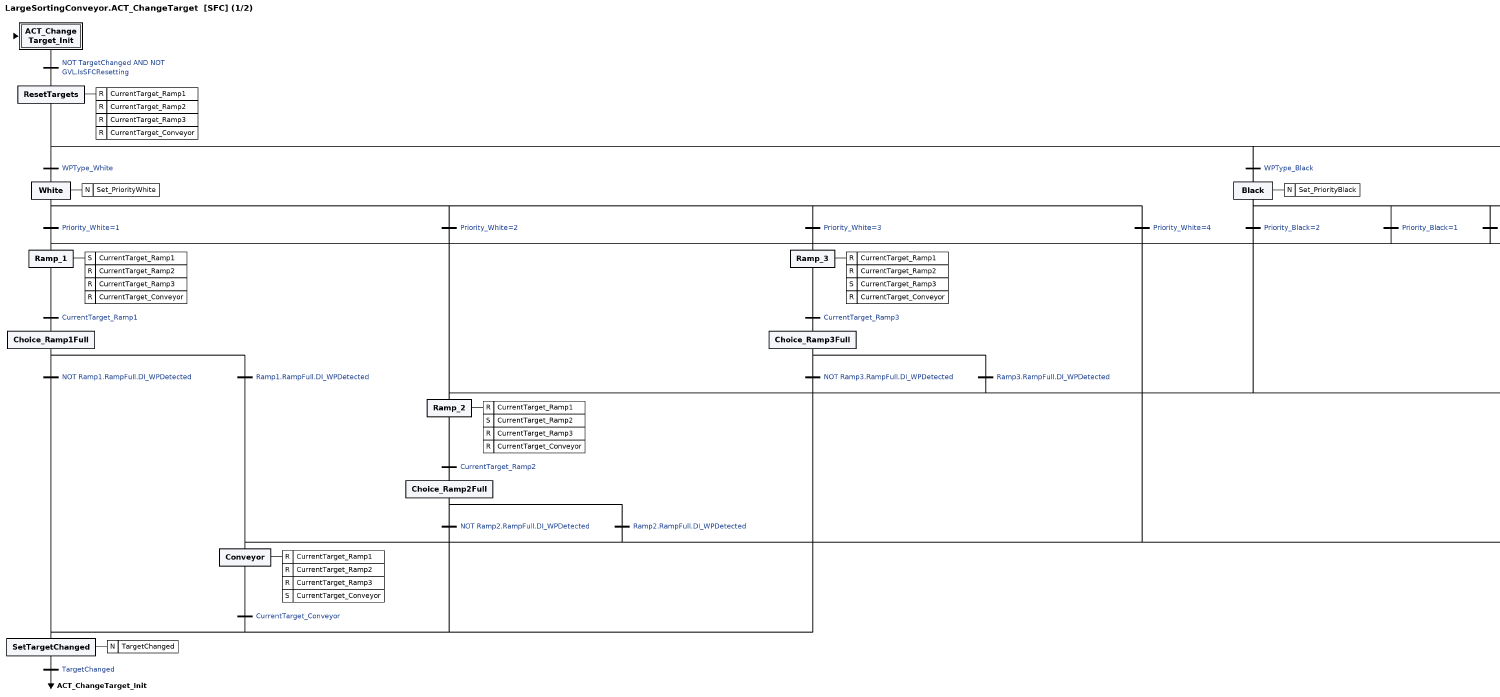
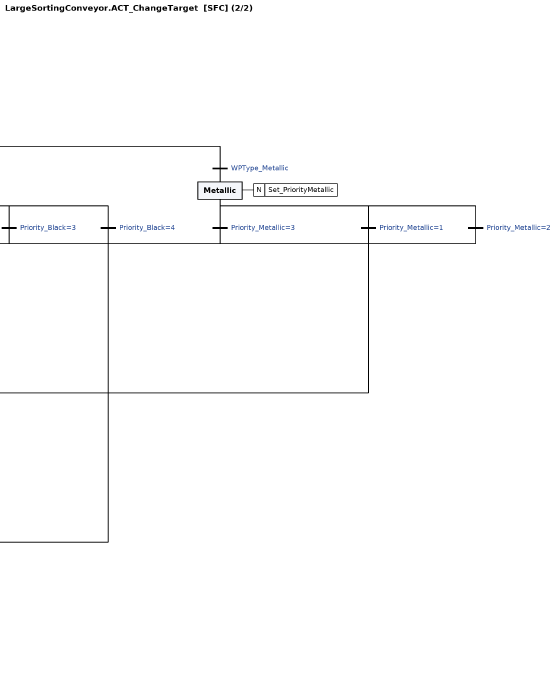
INITIAL_STEP ACT_ChangeTarget_Init:
END_STEP
TRANSITION FROM ACT_ChangeTarget_Init TO ResetTargets
  := NOT TargetChanged AND NOT GVL.IsSFCResetting;
END_TRANSITION
STEP ResetTargets:
  CurrentTarget_Ramp1(R);
  CurrentTarget_Ramp2(R);
  CurrentTarget_Ramp3(R);
  CurrentTarget_Conveyor(R);
END_STEP
TRANSITION FROM ResetTargets TO White
  := WPType_White;
END_TRANSITION
TRANSITION FROM ResetTargets TO Black
  := WPType_Black;
END_TRANSITION
TRANSITION FROM ResetTargets TO Metallic
  := WPType_Metallic;
END_TRANSITION
STEP White:
  Set_PriorityWhite(N);
END_STEP
TRANSITION FROM White TO Ramp_1
  := Priority_White=1;
END_TRANSITION
TRANSITION FROM White TO Ramp_2
  := Priority_White=2;
END_TRANSITION
TRANSITION FROM White TO Ramp_3
  := Priority_White=3;
END_TRANSITION
TRANSITION FROM White TO Conveyor
  := Priority_White=4;
END_TRANSITION
STEP Ramp_1:
  CurrentTarget_Ramp1(S);
  CurrentTarget_Ramp2(R);
  CurrentTarget_Ramp3(R);
  CurrentTarget_Conveyor(R);
END_STEP
TRANSITION FROM Ramp_1 TO Choice_Ramp1Full
  := CurrentTarget_Ramp1;
END_TRANSITION
STEP Choice_Ramp1Full:
END_STEP
TRANSITION FROM Choice_Ramp1Full TO SetTargetChanged
  := NOT Ramp1.RampFull.DI_WPDetected;
END_TRANSITION
TRANSITION FROM Choice_Ramp1Full TO Conveyor
  := Ramp1.RampFull.DI_WPDetected;
END_TRANSITION
STEP Conveyor:
  CurrentTarget_Ramp1(R);
  CurrentTarget_Ramp2(R);
  CurrentTarget_Ramp3(R);
  CurrentTarget_Conveyor(S);
END_STEP
TRANSITION FROM Conveyor TO SetTargetChanged
  := CurrentTarget_Conveyor;
END_TRANSITION
STEP Black:
  Set_PriorityBlack(N);
END_STEP
TRANSITION FROM Black TO Ramp_2
  := Priority_Black=2;
END_TRANSITION
TRANSITION FROM Black TO Ramp_1
  := Priority_Black=1;
END_TRANSITION
TRANSITION FROM Black TO Ramp_3
  := Priority_Black=3;
END_TRANSITION
TRANSITION FROM Black TO Conveyor
  := Priority_Black=4;
END_TRANSITION
STEP Ramp_2:
  CurrentTarget_Ramp1(R);
  CurrentTarget_Ramp2(S);
  CurrentTarget_Ramp3(R);
  CurrentTarget_Conveyor(R);
END_STEP
TRANSITION FROM Ramp_2 TO Choice_Ramp2Full
  := CurrentTarget_Ramp2;
END_TRANSITION
STEP Choice_Ramp2Full:
END_STEP
TRANSITION FROM Choice_Ramp2Full TO SetTargetChanged
  := NOT Ramp2.RampFull.DI_WPDetected;
END_TRANSITION
TRANSITION FROM Choice_Ramp2Full TO Conveyor
  := Ramp2.RampFull.DI_WPDetected;
END_TRANSITION
STEP Metallic:
  Set_PriorityMetallic(N);
END_STEP
TRANSITION FROM Metallic TO Ramp_3
  := Priority_Metallic=3;
END_TRANSITION
TRANSITION FROM Metallic TO Ramp_2
  := Priority_Metallic=1;
END_TRANSITION
TRANSITION FROM Metallic TO Ramp_3
  := Priority_Metallic=2;
END_TRANSITION
STEP Ramp_3:
  CurrentTarget_Ramp1(R);
  CurrentTarget_Ramp2(R);
  CurrentTarget_Ramp3(S);
  CurrentTarget_Conveyor(R);
END_STEP
TRANSITION FROM Ramp_3 TO Choice_Ramp3Full
  := CurrentTarget_Ramp3;
END_TRANSITION
STEP Choice_Ramp3Full:
END_STEP
TRANSITION FROM Choice_Ramp3Full TO SetTargetChanged
  := NOT Ramp3.RampFull.DI_WPDetected;
END_TRANSITION
TRANSITION FROM Choice_Ramp3Full TO Ramp_2
  := Ramp3.RampFull.DI_WPDetected;
END_TRANSITION
STEP SetTargetChanged:
  TargetChanged(N);
END_STEP
TRANSITION FROM SetTargetChanged TO ACT_ChangeTarget_Init
  := TargetChanged;
END_TRANSITION
END_ACTION

ACTION ACT_CheckWPType:
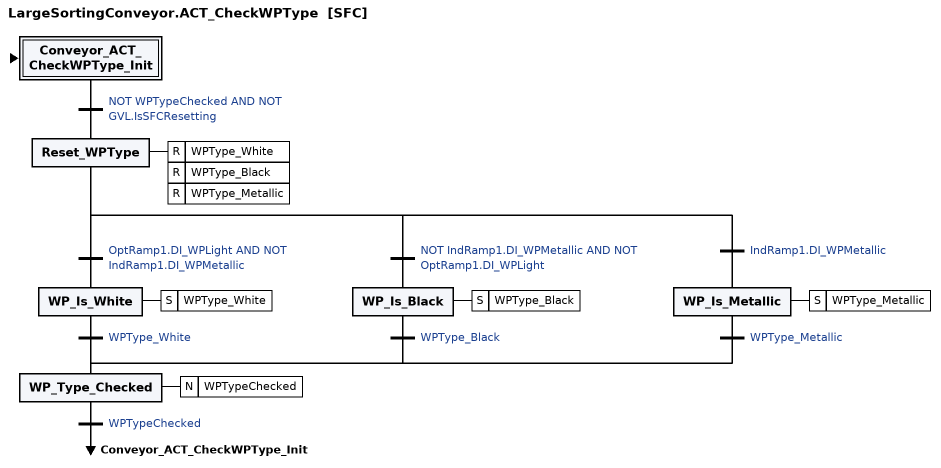
INITIAL_STEP Conveyor_ACT_CheckWPType_Init:
END_STEP
TRANSITION FROM Conveyor_ACT_CheckWPType_Init TO Reset_WPType
  := NOT WPTypeChecked AND NOT GVL.IsSFCResetting;
END_TRANSITION
STEP Reset_WPType:
  WPType_White(R);
  WPType_Black(R);
  WPType_Metallic(R);
END_STEP
TRANSITION FROM Reset_WPType TO WP_Is_White
  := OptRamp1.DI_WPLight AND NOT IndRamp1.DI_WPMetallic;
END_TRANSITION
TRANSITION FROM Reset_WPType TO WP_Is_Black
  := NOT IndRamp1.DI_WPMetallic AND NOT OptRamp1.DI_WPLight;
END_TRANSITION
TRANSITION FROM Reset_WPType TO WP_Is_Metallic
  := IndRamp1.DI_WPMetallic;
END_TRANSITION
STEP WP_Is_White:
  WPType_White(S);
END_STEP
TRANSITION FROM WP_Is_White TO WP_Type_Checked
  := WPType_White;
END_TRANSITION
STEP WP_Is_Black:
  WPType_Black(S);
END_STEP
TRANSITION FROM WP_Is_Black TO WP_Type_Checked
  := WPType_Black;
END_TRANSITION
STEP WP_Is_Metallic:
  WPType_Metallic(S);
END_STEP
TRANSITION FROM WP_Is_Metallic TO WP_Type_Checked
  := WPType_Metallic;
END_TRANSITION
STEP WP_Type_Checked:
  WPTypeChecked(N);
END_STEP
TRANSITION FROM WP_Type_Checked TO Conveyor_ACT_CheckWPType_Init
  := WPTypeChecked;
END_TRANSITION
END_ACTION

ACTION ACT_CountWPsAtConveyor:
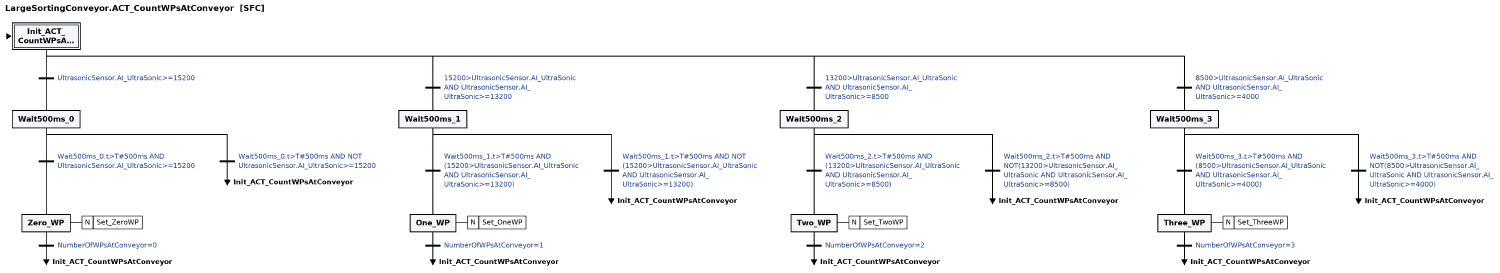
INITIAL_STEP Init_ACT_CountWPsAtConveyor:
END_STEP
TRANSITION FROM Init_ACT_CountWPsAtConveyor TO Wait500ms_0
  := UltrasonicSensor.AI_UltraSonic>=15200;
END_TRANSITION
TRANSITION FROM Init_ACT_CountWPsAtConveyor TO Wait500ms_1
  := 15200>UltrasonicSensor.AI_UltraSonic AND UltrasonicSensor.AI_UltraSonic>=13200;
END_TRANSITION
TRANSITION FROM Init_ACT_CountWPsAtConveyor TO Wait500ms_2
  := 13200>UltrasonicSensor.AI_UltraSonic AND UltrasonicSensor.AI_UltraSonic>=8500;
END_TRANSITION
TRANSITION FROM Init_ACT_CountWPsAtConveyor TO Wait500ms_3
  := 8500>UltrasonicSensor.AI_UltraSonic AND UltrasonicSensor.AI_UltraSonic>=4000;
END_TRANSITION
STEP Wait500ms_0:
END_STEP
TRANSITION FROM Wait500ms_0 TO Zero_WP
  := Wait500ms_0.t>T#500ms AND UltrasonicSensor.AI_UltraSonic>=15200;
END_TRANSITION
TRANSITION FROM Wait500ms_0 TO Init_ACT_CountWPsAtConveyor
  := Wait500ms_0.t>T#500ms AND NOT UltrasonicSensor.AI_UltraSonic>=15200;
END_TRANSITION
STEP Zero_WP:
  Set_ZeroWP(N);
END_STEP
TRANSITION FROM Zero_WP TO Init_ACT_CountWPsAtConveyor
  := NumberOfWPsAtConveyor=0;
END_TRANSITION
STEP Wait500ms_1:
END_STEP
TRANSITION FROM Wait500ms_1 TO One_WP
  := Wait500ms_1.t>T#500ms AND (15200>UltrasonicSensor.AI_UltraSonic AND UltrasonicSensor.AI_UltraSonic>=13200);
END_TRANSITION
TRANSITION FROM Wait500ms_1 TO Init_ACT_CountWPsAtConveyor
  := Wait500ms_1.t>T#500ms AND NOT (15200>UltrasonicSensor.AI_UltraSonic AND UltrasonicSensor.AI_UltraSonic>=13200);
END_TRANSITION
STEP One_WP:
  Set_OneWP(N);
END_STEP
TRANSITION FROM One_WP TO Init_ACT_CountWPsAtConveyor
  := NumberOfWPsAtConveyor=1;
END_TRANSITION
STEP Wait500ms_2:
END_STEP
TRANSITION FROM Wait500ms_2 TO Two_WP
  := Wait500ms_2.t>T#500ms AND (13200>UltrasonicSensor.AI_UltraSonic AND UltrasonicSensor.AI_UltraSonic>=8500);
END_TRANSITION
TRANSITION FROM Wait500ms_2 TO Init_ACT_CountWPsAtConveyor
  := Wait500ms_2.t>T#500ms AND NOT(13200>UltrasonicSensor.AI_UltraSonic AND UltrasonicSensor.AI_UltraSonic>=8500);
END_TRANSITION
STEP Two_WP:
  Set_TwoWP(N);
END_STEP
TRANSITION FROM Two_WP TO Init_ACT_CountWPsAtConveyor
  := NumberOfWPsAtConveyor=2;
END_TRANSITION
STEP Wait500ms_3:
END_STEP
TRANSITION FROM Wait500ms_3 TO Three_WP
  := Wait500ms_3.t>T#500ms AND (8500>UltrasonicSensor.AI_UltraSonic AND UltrasonicSensor.AI_UltraSonic>=4000);
END_TRANSITION
TRANSITION FROM Wait500ms_3 TO Init_ACT_CountWPsAtConveyor
  := Wait500ms_3.t>T#500ms AND NOT(8500>UltrasonicSensor.AI_UltraSonic AND UltrasonicSensor.AI_UltraSonic>=4000);
END_TRANSITION
STEP Three_WP:
  Set_ThreeWP(N);
END_STEP
TRANSITION FROM Three_WP TO Init_ACT_CountWPsAtConveyor
  := NumberOfWPsAtConveyor=3;
END_TRANSITION
END_ACTION

ACTION ACT_SortWP:
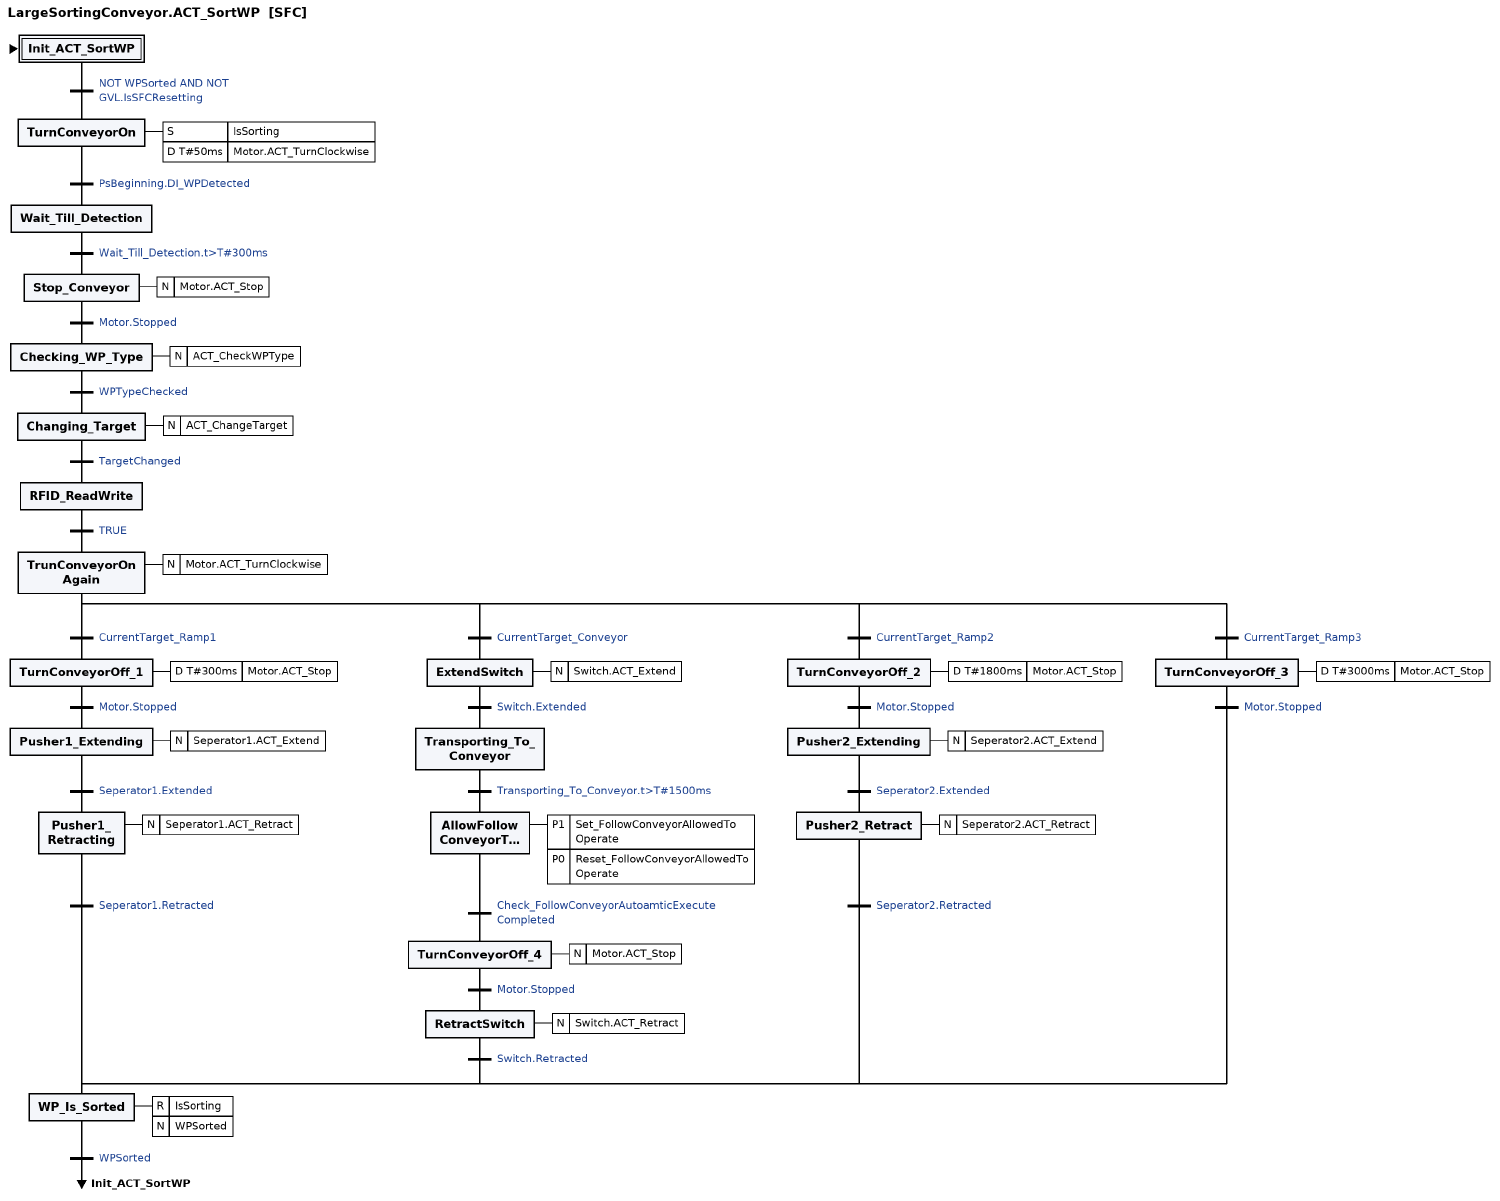
INITIAL_STEP Init_ACT_SortWP:
END_STEP
TRANSITION FROM Init_ACT_SortWP TO TurnConveyorOn
  := NOT WPSorted AND NOT GVL.IsSFCResetting;
END_TRANSITION
STEP TurnConveyorOn:
  IsSorting(S);
  Motor.ACT_TurnClockwise(D, T#50ms);
END_STEP
TRANSITION FROM TurnConveyorOn TO Wait_Till_Detection
  := PsBeginning.DI_WPDetected;
END_TRANSITION
STEP Wait_Till_Detection:
END_STEP
TRANSITION FROM Wait_Till_Detection TO Stop_Conveyor
  := Wait_Till_Detection.t>T#300ms;
END_TRANSITION
STEP Stop_Conveyor:
  Motor.ACT_Stop(N);
END_STEP
TRANSITION FROM Stop_Conveyor TO Checking_WP_Type
  := Motor.Stopped;
END_TRANSITION
STEP Checking_WP_Type:
  ACT_CheckWPType(N);
END_STEP
TRANSITION FROM Checking_WP_Type TO Changing_Target
  := WPTypeChecked;
END_TRANSITION
STEP Changing_Target:
  ACT_ChangeTarget(N);
END_STEP
TRANSITION FROM Changing_Target TO RFID_ReadWrite
  := TargetChanged;
END_TRANSITION
STEP RFID_ReadWrite:
END_STEP
TRANSITION FROM RFID_ReadWrite TO TrunConveyorOnAgain
  := TRUE;
END_TRANSITION
STEP TrunConveyorOnAgain:
  Motor.ACT_TurnClockwise(N);
END_STEP
TRANSITION FROM TrunConveyorOnAgain TO TurnConveyorOff_1
  := CurrentTarget_Ramp1;
END_TRANSITION
TRANSITION FROM TrunConveyorOnAgain TO ExtendSwitch
  := CurrentTarget_Conveyor;
END_TRANSITION
TRANSITION FROM TrunConveyorOnAgain TO TurnConveyorOff_2
  := CurrentTarget_Ramp2;
END_TRANSITION
TRANSITION FROM TrunConveyorOnAgain TO TurnConveyorOff_3
  := CurrentTarget_Ramp3;
END_TRANSITION
STEP TurnConveyorOff_1:
  Motor.ACT_Stop(D, T#300ms);
END_STEP
TRANSITION FROM TurnConveyorOff_1 TO Pusher1_Extending
  := Motor.Stopped;
END_TRANSITION
STEP Pusher1_Extending:
  Seperator1.ACT_Extend(N);
END_STEP
TRANSITION FROM Pusher1_Extending TO Pusher1_Retracting
  := Seperator1.Extended;
END_TRANSITION
STEP Pusher1_Retracting:
  Seperator1.ACT_Retract(N);
END_STEP
TRANSITION FROM Pusher1_Retracting TO WP_Is_Sorted
  := Seperator1.Retracted;
END_TRANSITION
STEP ExtendSwitch:
  Switch.ACT_Extend(N);
END_STEP
TRANSITION FROM ExtendSwitch TO Transporting_To_Conveyor
  := Switch.Extended;
END_TRANSITION
STEP Transporting_To_Conveyor:
END_STEP
TRANSITION FROM Transporting_To_Conveyor TO AllowFollowConveyorToReceiveWP
  := Transporting_To_Conveyor.t>T#1500ms;
END_TRANSITION
STEP AllowFollowConveyorToReceiveWP:
  Set_FollowConveyorAllowedToOperate(P1);
  Reset_FollowConveyorAllowedToOperate(P0);
END_STEP
TRANSITION FROM AllowFollowConveyorToReceiveWP TO TurnConveyorOff_4
  := Check_FollowConveyorAutoamticExecuteCompleted;
END_TRANSITION
STEP TurnConveyorOff_4:
  Motor.ACT_Stop(N);
END_STEP
TRANSITION FROM TurnConveyorOff_4 TO RetractSwitch
  := Motor.Stopped;
END_TRANSITION
STEP RetractSwitch:
  Switch.ACT_Retract(N);
END_STEP
TRANSITION FROM RetractSwitch TO WP_Is_Sorted
  := Switch.Retracted;
END_TRANSITION
STEP TurnConveyorOff_2:
  Motor.ACT_Stop(D, T#1800ms);
END_STEP
TRANSITION FROM TurnConveyorOff_2 TO Pusher2_Extending
  := Motor.Stopped;
END_TRANSITION
STEP Pusher2_Extending:
  Seperator2.ACT_Extend(N);
END_STEP
TRANSITION FROM Pusher2_Extending TO Pusher2_Retract
  := Seperator2.Extended;
END_TRANSITION
STEP Pusher2_Retract:
  Seperator2.ACT_Retract(N);
END_STEP
TRANSITION FROM Pusher2_Retract TO WP_Is_Sorted
  := Seperator2.Retracted;
END_TRANSITION
STEP TurnConveyorOff_3:
  Motor.ACT_Stop(D, T#3000ms);
END_STEP
TRANSITION FROM TurnConveyorOff_3 TO WP_Is_Sorted
  := Motor.Stopped;
END_TRANSITION
STEP WP_Is_Sorted:
  IsSorting(R);
  WPSorted(N);
END_STEP
TRANSITION FROM WP_Is_Sorted TO Init_ACT_SortWP
  := WPSorted;
END_TRANSITION
END_ACTION

ACTION ACT_AutomaticExecute:
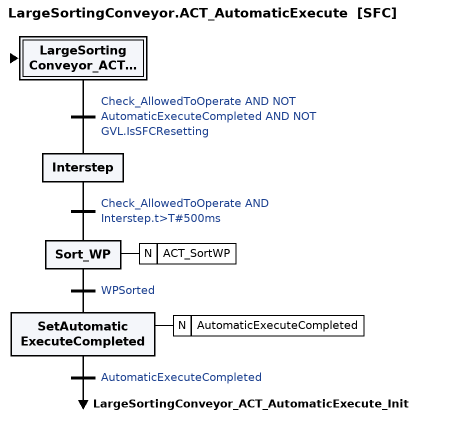
INITIAL_STEP LargeSortingConveyor_ACT_AutomaticExecute_Init:
END_STEP
TRANSITION FROM LargeSortingConveyor_ACT_AutomaticExecute_Init TO Interstep
  := Check_AllowedToOperate AND NOT AutomaticExecuteCompleted AND NOT GVL.IsSFCResetting;
END_TRANSITION
STEP Interstep:
END_STEP
TRANSITION FROM Interstep TO Sort_WP
  := Check_AllowedToOperate AND Interstep.t>T#500ms;
END_TRANSITION
STEP Sort_WP:
  ACT_SortWP(N);
END_STEP
TRANSITION FROM Sort_WP TO SetAutomaticExecuteCompleted
  := WPSorted;
END_TRANSITION
STEP SetAutomaticExecuteCompleted:
  AutomaticExecuteCompleted(N);
END_STEP
TRANSITION FROM SetAutomaticExecuteCompleted TO LargeSortingConveyor_ACT_AutomaticExecute_Init
  := AutomaticExecuteCompleted;
END_TRANSITION
END_ACTION

ACTION ACT_EmergencyStop:
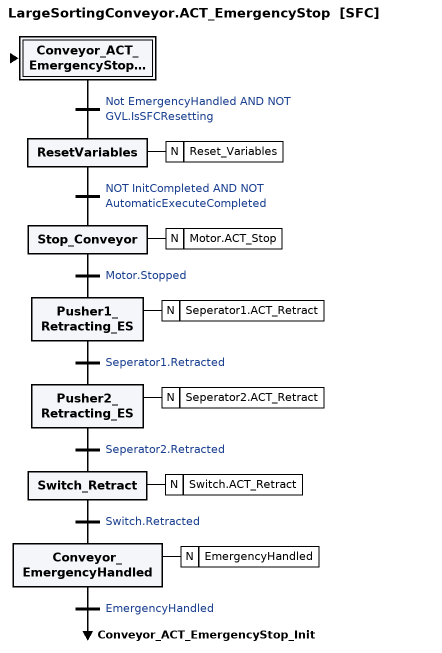
INITIAL_STEP Conveyor_ACT_EmergencyStop_Init:
END_STEP
TRANSITION FROM Conveyor_ACT_EmergencyStop_Init TO ResetVariables
  := Not EmergencyHandled AND NOT GVL.IsSFCResetting;
END_TRANSITION
STEP ResetVariables:
  Reset_Variables(N);
END_STEP
TRANSITION FROM ResetVariables TO Stop_Conveyor
  := NOT InitCompleted AND NOT AutomaticExecuteCompleted;
END_TRANSITION
STEP Stop_Conveyor:
  Motor.ACT_Stop(N);
END_STEP
TRANSITION FROM Stop_Conveyor TO Pusher1_Retracting_ES
  := Motor.Stopped;
END_TRANSITION
STEP Pusher1_Retracting_ES:
  Seperator1.ACT_Retract(N);
END_STEP
TRANSITION FROM Pusher1_Retracting_ES TO Pusher2_Retracting_ES
  := Seperator1.Retracted;
END_TRANSITION
STEP Pusher2_Retracting_ES:
  Seperator2.ACT_Retract(N);
END_STEP
TRANSITION FROM Pusher2_Retracting_ES TO Switch_Retract
  := Seperator2.Retracted;
END_TRANSITION
STEP Switch_Retract:
  Switch.ACT_Retract(N);
END_STEP
TRANSITION FROM Switch_Retract TO Conveyor_EmergencyHandled
  := Switch.Retracted;
END_TRANSITION
STEP Conveyor_EmergencyHandled:
  EmergencyHandled(N);
END_STEP
TRANSITION FROM Conveyor_EmergencyHandled TO Conveyor_ACT_EmergencyStop_Init
  := EmergencyHandled;
END_TRANSITION
END_ACTION

ACTION ACT_Init:
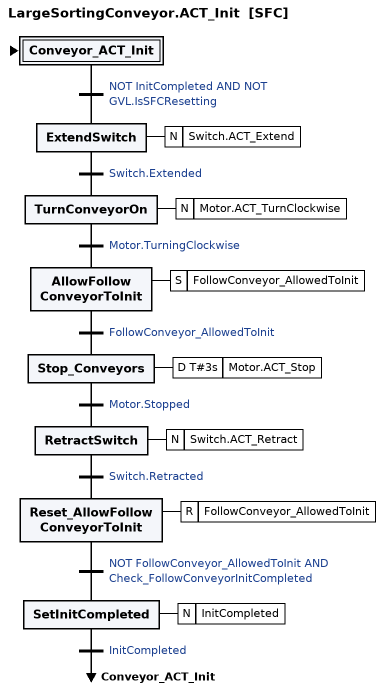
INITIAL_STEP Conveyor_ACT_Init:
END_STEP
TRANSITION FROM Conveyor_ACT_Init TO ExtendSwitch
  := NOT InitCompleted AND NOT GVL.IsSFCResetting;
END_TRANSITION
STEP ExtendSwitch:
  Switch.ACT_Extend(N);
END_STEP
TRANSITION FROM ExtendSwitch TO TurnConveyorOn
  := Switch.Extended;
END_TRANSITION
STEP TurnConveyorOn:
  Motor.ACT_TurnClockwise(N);
END_STEP
TRANSITION FROM TurnConveyorOn TO AllowFollowConveyorToInit
  := Motor.TurningClockwise;
END_TRANSITION
STEP AllowFollowConveyorToInit:
  FollowConveyor_AllowedToInit(S);
END_STEP
TRANSITION FROM AllowFollowConveyorToInit TO Stop_Conveyors
  := FollowConveyor_AllowedToInit;
END_TRANSITION
STEP Stop_Conveyors:
  Motor.ACT_Stop(D, T#3s);
END_STEP
TRANSITION FROM Stop_Conveyors TO RetractSwitch
  := Motor.Stopped;
END_TRANSITION
STEP RetractSwitch:
  Switch.ACT_Retract(N);
END_STEP
TRANSITION FROM RetractSwitch TO Reset_AllowFollowConveyorToInit
  := Switch.Retracted;
END_TRANSITION
STEP Reset_AllowFollowConveyorToInit:
  FollowConveyor_AllowedToInit(R);
END_STEP
TRANSITION FROM Reset_AllowFollowConveyorToInit TO SetInitCompleted
  := NOT FollowConveyor_AllowedToInit AND Check_FollowConveyorInitCompleted;
END_TRANSITION
STEP SetInitCompleted:
  InitCompleted(N);
END_STEP
TRANSITION FROM SetInitCompleted TO Conveyor_ACT_Init
  := InitCompleted;
END_TRANSITION
END_ACTION
END_FUNCTION_BLOCK

FUNCTION_BLOCK PicAlpha
VAR_INPUT
	//Hardware
	AtPosition1 : PositionTransmitter;
	AtPosition2 : PositionTransmitter;
	AtPosition3 : PositionTransmitter; 
	AtPosition4 : PositionTransmitter;
	Motor : Motor;
	Gripper : VacuumGripperExtended;
	LiftingCylinder : MonostableCylinder;
	
	//Software
	SoftwareEmergency : BOOL;
	Check_AllowedToOperate : BOOL;
	Check_Conveyor_AutomaticExecuteCompleted : BOOL;
	Check_EngineStop : BOOL;
	SFCReset : BOOL; //Only for SFC
END_VAR
VAR_OUTPUT
	//Software
	InitCompleted : BOOL;
	Conveyor_AllowedToOperate : BOOL;
	AutomaticExecuteCompleted : BOOL;
	EmergencyHandled : BOOL;	
END_VAR
VAR
	WPPickedUp : BOOL;
	WPPutDown : BOOL;
	ReachedPosition1 : BOOL;
	ReachedPosition2 : BOOL;
	ReachedPosition3 : BOOL;
	ReachedPosition4 : BOOL;
END_VAR

                  Check_AllowedToOperate := MAIN.Check_PicAlpha_AllowedToOperate;
Check_Conveyor_AutomaticExecuteCompleted := MAIN.Check_PicAlpha_Conveyor_AutomaticExecuteCompleted;
Check_EngineStop := MAIN.PPU_EngineStop;
IF Check_EngineStop THEN
	Motor.ACT_Stop();
END_IF
                

ACTION Reset_Variables:
                      InitCompleted := FALSE;
Conveyor_AllowedToOperate := FALSE;
AutomaticExecuteCompleted := FALSE;

WPPickedUp := FALSE;
WPPutDown := FALSE;
ReachedPosition1 := FALSE;
ReachedPosition2 := FALSE;
ReachedPosition3 := FALSE;
ReachedPosition4 := FALSE;
                    
END_ACTION

ACTION ACT_MoveToPos1:
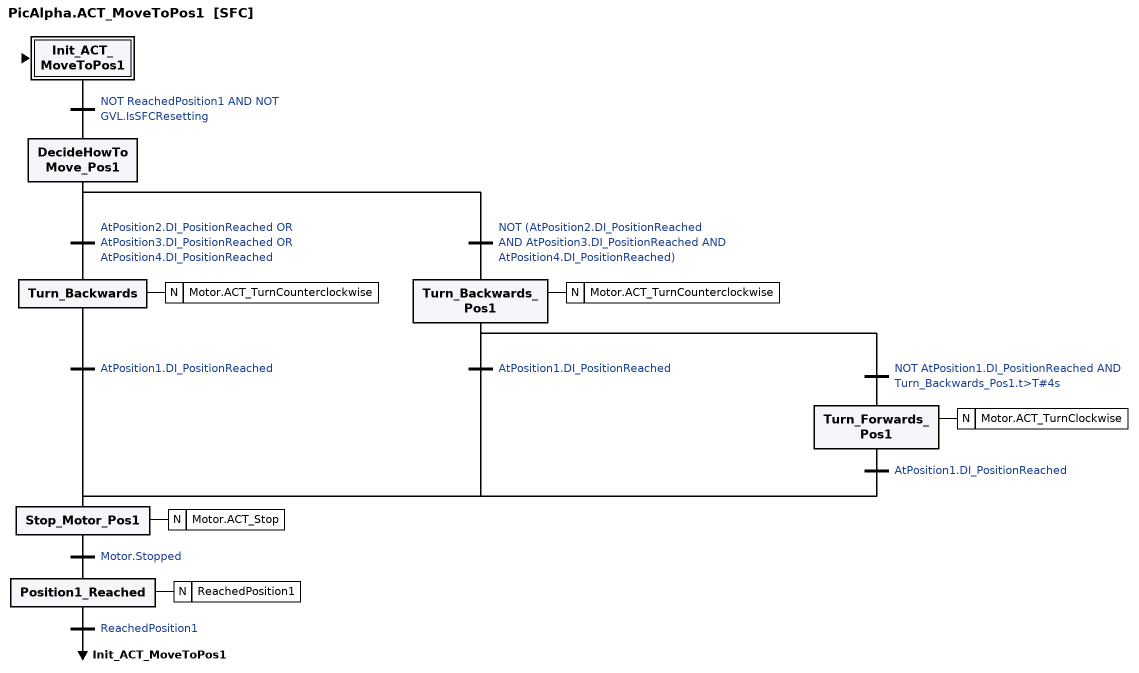
INITIAL_STEP Init_ACT_MoveToPos1:
END_STEP
TRANSITION FROM Init_ACT_MoveToPos1 TO DecideHowToMove_Pos1
  := NOT ReachedPosition1 AND NOT GVL.IsSFCResetting;
END_TRANSITION
STEP DecideHowToMove_Pos1:
END_STEP
TRANSITION FROM DecideHowToMove_Pos1 TO Turn_Backwards
  := AtPosition2.DI_PositionReached OR AtPosition3.DI_PositionReached OR AtPosition4.DI_PositionReached;
END_TRANSITION
TRANSITION FROM DecideHowToMove_Pos1 TO Turn_Backwards_Pos1
  := NOT (AtPosition2.DI_PositionReached AND AtPosition3.DI_PositionReached AND AtPosition4.DI_PositionReached);
END_TRANSITION
STEP Turn_Backwards:
  Motor.ACT_TurnCounterclockwise(N);
END_STEP
TRANSITION FROM Turn_Backwards TO Stop_Motor_Pos1
  := AtPosition1.DI_PositionReached;
END_TRANSITION
STEP Turn_Backwards_Pos1:
  Motor.ACT_TurnCounterclockwise(N);
END_STEP
TRANSITION FROM Turn_Backwards_Pos1 TO Stop_Motor_Pos1
  := AtPosition1.DI_PositionReached;
END_TRANSITION
TRANSITION FROM Turn_Backwards_Pos1 TO Turn_Forwards_Pos1
  := NOT AtPosition1.DI_PositionReached AND Turn_Backwards_Pos1.t>T#4s;
END_TRANSITION
STEP Turn_Forwards_Pos1:
  Motor.ACT_TurnClockwise(N);
END_STEP
TRANSITION FROM Turn_Forwards_Pos1 TO Stop_Motor_Pos1
  := AtPosition1.DI_PositionReached;
END_TRANSITION
STEP Stop_Motor_Pos1:
  Motor.ACT_Stop(N);
END_STEP
TRANSITION FROM Stop_Motor_Pos1 TO Position1_Reached
  := Motor.Stopped;
END_TRANSITION
STEP Position1_Reached:
  ReachedPosition1(N);
END_STEP
TRANSITION FROM Position1_Reached TO Init_ACT_MoveToPos1
  := ReachedPosition1;
END_TRANSITION
END_ACTION

ACTION ACT_MoveToPos2:
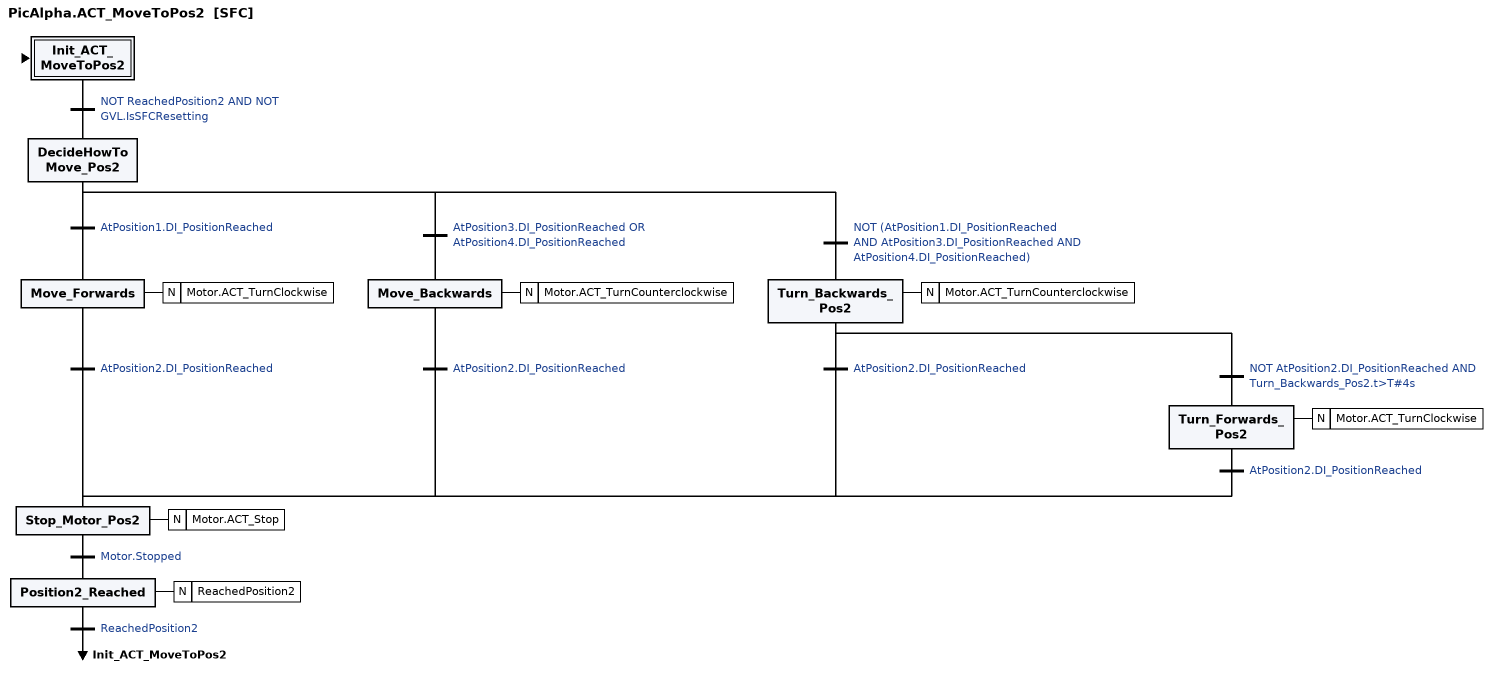
INITIAL_STEP Init_ACT_MoveToPos2:
END_STEP
TRANSITION FROM Init_ACT_MoveToPos2 TO DecideHowToMove_Pos2
  := NOT ReachedPosition2 AND NOT GVL.IsSFCResetting;
END_TRANSITION
STEP DecideHowToMove_Pos2:
END_STEP
TRANSITION FROM DecideHowToMove_Pos2 TO Move_Forwards
  := AtPosition1.DI_PositionReached;
END_TRANSITION
TRANSITION FROM DecideHowToMove_Pos2 TO Move_Backwards
  := AtPosition3.DI_PositionReached OR AtPosition4.DI_PositionReached;
END_TRANSITION
TRANSITION FROM DecideHowToMove_Pos2 TO Turn_Backwards_Pos2
  := NOT (AtPosition1.DI_PositionReached AND AtPosition3.DI_PositionReached AND AtPosition4.DI_PositionReached);
END_TRANSITION
STEP Move_Forwards:
  Motor.ACT_TurnClockwise(N);
END_STEP
TRANSITION FROM Move_Forwards TO Stop_Motor_Pos2
  := AtPosition2.DI_PositionReached;
END_TRANSITION
STEP Move_Backwards:
  Motor.ACT_TurnCounterclockwise(N);
END_STEP
TRANSITION FROM Move_Backwards TO Stop_Motor_Pos2
  := AtPosition2.DI_PositionReached;
END_TRANSITION
STEP Turn_Backwards_Pos2:
  Motor.ACT_TurnCounterclockwise(N);
END_STEP
TRANSITION FROM Turn_Backwards_Pos2 TO Stop_Motor_Pos2
  := AtPosition2.DI_PositionReached;
END_TRANSITION
TRANSITION FROM Turn_Backwards_Pos2 TO Turn_Forwards_Pos2
  := NOT AtPosition2.DI_PositionReached AND Turn_Backwards_Pos2.t>T#4s;
END_TRANSITION
STEP Turn_Forwards_Pos2:
  Motor.ACT_TurnClockwise(N);
END_STEP
TRANSITION FROM Turn_Forwards_Pos2 TO Stop_Motor_Pos2
  := AtPosition2.DI_PositionReached;
END_TRANSITION
STEP Stop_Motor_Pos2:
  Motor.ACT_Stop(N);
END_STEP
TRANSITION FROM Stop_Motor_Pos2 TO Position2_Reached
  := Motor.Stopped;
END_TRANSITION
STEP Position2_Reached:
  ReachedPosition2(N);
END_STEP
TRANSITION FROM Position2_Reached TO Init_ACT_MoveToPos2
  := ReachedPosition2;
END_TRANSITION
END_ACTION

ACTION ACT_MoveToPos3:
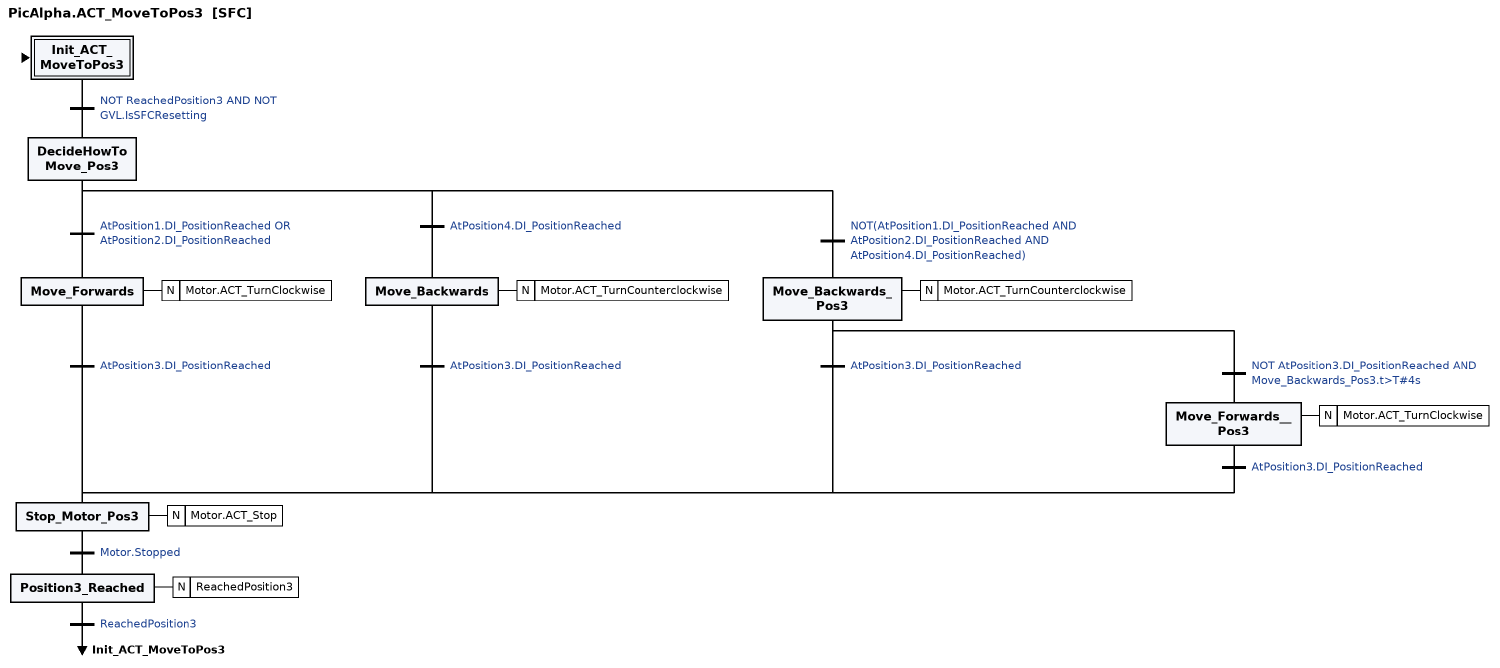
INITIAL_STEP Init_ACT_MoveToPos3:
END_STEP
TRANSITION FROM Init_ACT_MoveToPos3 TO DecideHowToMove_Pos3
  := NOT ReachedPosition3 AND NOT GVL.IsSFCResetting;
END_TRANSITION
STEP DecideHowToMove_Pos3:
END_STEP
TRANSITION FROM DecideHowToMove_Pos3 TO Move_Forwards
  := AtPosition1.DI_PositionReached OR AtPosition2.DI_PositionReached;
END_TRANSITION
TRANSITION FROM DecideHowToMove_Pos3 TO Move_Backwards
  := AtPosition4.DI_PositionReached;
END_TRANSITION
TRANSITION FROM DecideHowToMove_Pos3 TO Move_Backwards_Pos3
  := NOT(AtPosition1.DI_PositionReached AND AtPosition2.DI_PositionReached AND AtPosition4.DI_PositionReached);
END_TRANSITION
STEP Move_Forwards:
  Motor.ACT_TurnClockwise(N);
END_STEP
TRANSITION FROM Move_Forwards TO Stop_Motor_Pos3
  := AtPosition3.DI_PositionReached;
END_TRANSITION
STEP Move_Backwards:
  Motor.ACT_TurnCounterclockwise(N);
END_STEP
TRANSITION FROM Move_Backwards TO Stop_Motor_Pos3
  := AtPosition3.DI_PositionReached;
END_TRANSITION
STEP Move_Backwards_Pos3:
  Motor.ACT_TurnCounterclockwise(N);
END_STEP
TRANSITION FROM Move_Backwards_Pos3 TO Stop_Motor_Pos3
  := AtPosition3.DI_PositionReached;
END_TRANSITION
TRANSITION FROM Move_Backwards_Pos3 TO Move_Forwards__Pos3
  := NOT AtPosition3.DI_PositionReached AND Move_Backwards_Pos3.t>T#4s;
END_TRANSITION
STEP Move_Forwards__Pos3:
  Motor.ACT_TurnClockwise(N);
END_STEP
TRANSITION FROM Move_Forwards__Pos3 TO Stop_Motor_Pos3
  := AtPosition3.DI_PositionReached;
END_TRANSITION
STEP Stop_Motor_Pos3:
  Motor.ACT_Stop(N);
END_STEP
TRANSITION FROM Stop_Motor_Pos3 TO Position3_Reached
  := Motor.Stopped;
END_TRANSITION
STEP Position3_Reached:
  ReachedPosition3(N);
END_STEP
TRANSITION FROM Position3_Reached TO Init_ACT_MoveToPos3
  := ReachedPosition3;
END_TRANSITION
END_ACTION

ACTION ACT_MoveToPos4:
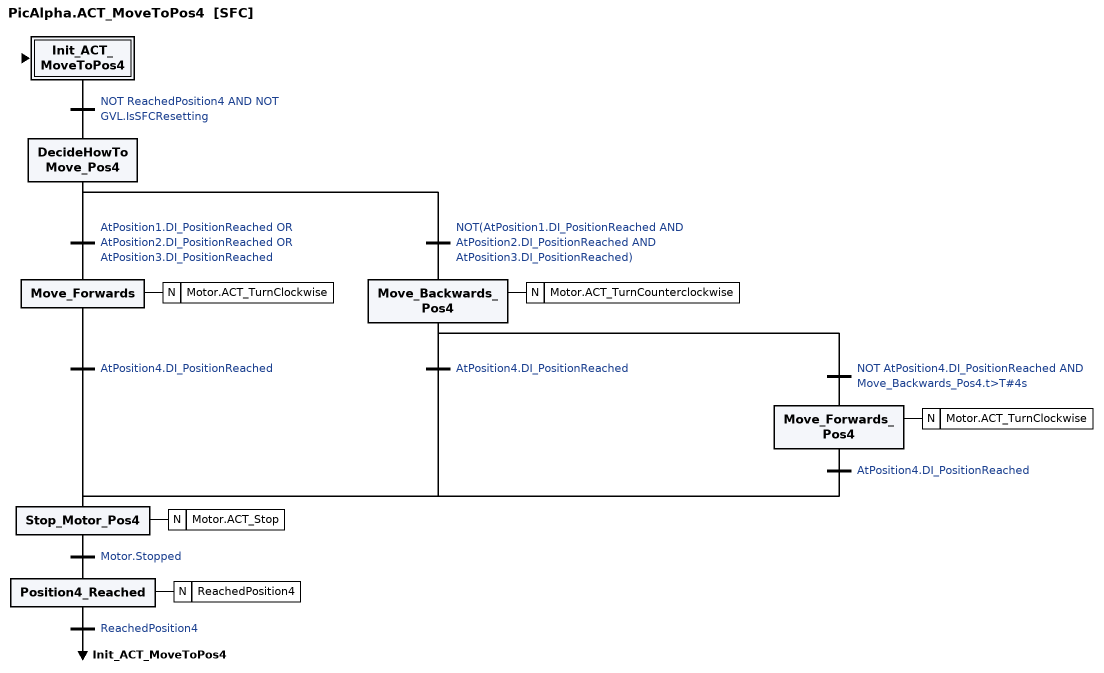
INITIAL_STEP Init_ACT_MoveToPos4:
END_STEP
TRANSITION FROM Init_ACT_MoveToPos4 TO DecideHowToMove_Pos4
  := NOT ReachedPosition4 AND NOT GVL.IsSFCResetting;
END_TRANSITION
STEP DecideHowToMove_Pos4:
END_STEP
TRANSITION FROM DecideHowToMove_Pos4 TO Move_Forwards
  := AtPosition1.DI_PositionReached OR AtPosition2.DI_PositionReached OR AtPosition3.DI_PositionReached;
END_TRANSITION
TRANSITION FROM DecideHowToMove_Pos4 TO Move_Backwards_Pos4
  := NOT(AtPosition1.DI_PositionReached AND AtPosition2.DI_PositionReached AND AtPosition3.DI_PositionReached);
END_TRANSITION
STEP Move_Forwards:
  Motor.ACT_TurnClockwise(N);
END_STEP
TRANSITION FROM Move_Forwards TO Stop_Motor_Pos4
  := AtPosition4.DI_PositionReached;
END_TRANSITION
STEP Move_Backwards_Pos4:
  Motor.ACT_TurnCounterclockwise(N);
END_STEP
TRANSITION FROM Move_Backwards_Pos4 TO Stop_Motor_Pos4
  := AtPosition4.DI_PositionReached;
END_TRANSITION
TRANSITION FROM Move_Backwards_Pos4 TO Move_Forwards_Pos4
  := NOT AtPosition4.DI_PositionReached AND Move_Backwards_Pos4.t>T#4s;
END_TRANSITION
STEP Move_Forwards_Pos4:
  Motor.ACT_TurnClockwise(N);
END_STEP
TRANSITION FROM Move_Forwards_Pos4 TO Stop_Motor_Pos4
  := AtPosition4.DI_PositionReached;
END_TRANSITION
STEP Stop_Motor_Pos4:
  Motor.ACT_Stop(N);
END_STEP
TRANSITION FROM Stop_Motor_Pos4 TO Position4_Reached
  := Motor.Stopped;
END_TRANSITION
STEP Position4_Reached:
  ReachedPosition4(N);
END_STEP
TRANSITION FROM Position4_Reached TO Init_ACT_MoveToPos4
  := ReachedPosition4;
END_TRANSITION
END_ACTION

ACTION ACT_PickUpWP:
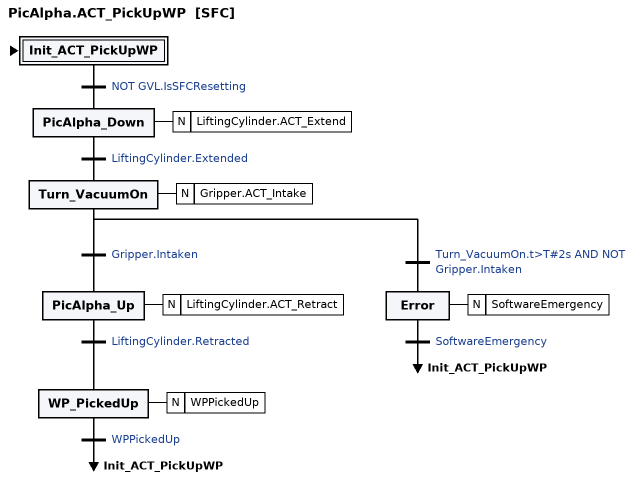
INITIAL_STEP Init_ACT_PickUpWP:
END_STEP
TRANSITION FROM Init_ACT_PickUpWP TO PicAlpha_Down
  := NOT GVL.IsSFCResetting;
END_TRANSITION
STEP PicAlpha_Down:
  LiftingCylinder.ACT_Extend(N);
END_STEP
TRANSITION FROM PicAlpha_Down TO Turn_VacuumOn
  := LiftingCylinder.Extended;
END_TRANSITION
STEP Turn_VacuumOn:
  Gripper.ACT_Intake(N);
END_STEP
TRANSITION FROM Turn_VacuumOn TO PicAlpha_Up
  := Gripper.Intaken;
END_TRANSITION
TRANSITION FROM Turn_VacuumOn TO Error
  := Turn_VacuumOn.t>T#2s AND NOT Gripper.Intaken;
END_TRANSITION
STEP PicAlpha_Up:
  LiftingCylinder.ACT_Retract(N);
END_STEP
TRANSITION FROM PicAlpha_Up TO WP_PickedUp
  := LiftingCylinder.Retracted;
END_TRANSITION
STEP WP_PickedUp:
  WPPickedUp(N);
END_STEP
TRANSITION FROM WP_PickedUp TO Init_ACT_PickUpWP
  := WPPickedUp;
END_TRANSITION
STEP Error:
  SoftwareEmergency(N);
END_STEP
TRANSITION FROM Error TO Init_ACT_PickUpWP
  := SoftwareEmergency;
END_TRANSITION
END_ACTION

ACTION ACT_PutDownWP:
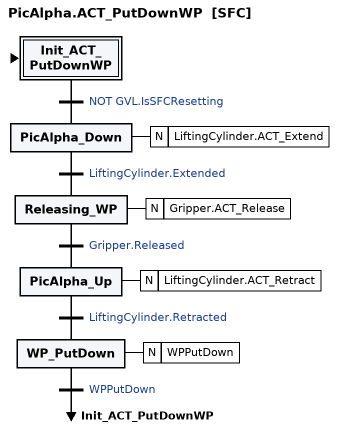
INITIAL_STEP Init_ACT_PutDownWP:
END_STEP
TRANSITION FROM Init_ACT_PutDownWP TO PicAlpha_Down
  := NOT GVL.IsSFCResetting;
END_TRANSITION
STEP PicAlpha_Down:
  LiftingCylinder.ACT_Extend(N);
END_STEP
TRANSITION FROM PicAlpha_Down TO Releasing_WP
  := LiftingCylinder.Extended;
END_TRANSITION
STEP Releasing_WP:
  Gripper.ACT_Release(N);
END_STEP
TRANSITION FROM Releasing_WP TO PicAlpha_Up
  := Gripper.Released;
END_TRANSITION
STEP PicAlpha_Up:
  LiftingCylinder.ACT_Retract(N);
END_STEP
TRANSITION FROM PicAlpha_Up TO WP_PutDown
  := LiftingCylinder.Retracted;
END_TRANSITION
STEP WP_PutDown:
  WPPutDown(N);
END_STEP
TRANSITION FROM WP_PutDown TO Init_ACT_PutDownWP
  := WPPutDown;
END_TRANSITION
END_ACTION

ACTION ACT_AutomaticExecute:
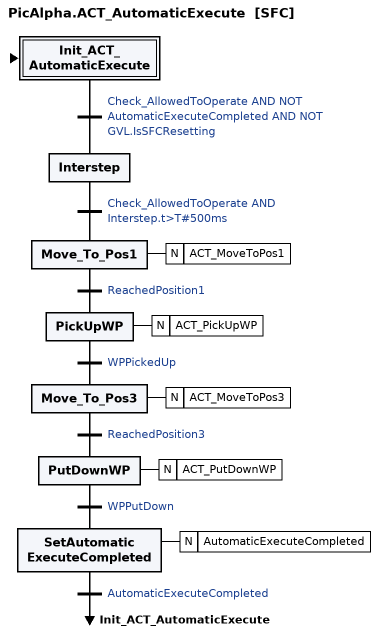
INITIAL_STEP Init_ACT_AutomaticExecute:
END_STEP
TRANSITION FROM Init_ACT_AutomaticExecute TO Interstep
  := Check_AllowedToOperate AND NOT AutomaticExecuteCompleted AND NOT GVL.IsSFCResetting;
END_TRANSITION
STEP Interstep:
END_STEP
TRANSITION FROM Interstep TO Move_To_Pos1
  := Check_AllowedToOperate AND Interstep.t>T#500ms;
END_TRANSITION
STEP Move_To_Pos1:
  ACT_MoveToPos1(N);
END_STEP
TRANSITION FROM Move_To_Pos1 TO PickUpWP
  := ReachedPosition1;
END_TRANSITION
STEP PickUpWP:
  ACT_PickUpWP(N);
END_STEP
TRANSITION FROM PickUpWP TO Move_To_Pos3
  := WPPickedUp;
END_TRANSITION
STEP Move_To_Pos3:
  ACT_MoveToPos3(N);
END_STEP
TRANSITION FROM Move_To_Pos3 TO PutDownWP
  := ReachedPosition3;
END_TRANSITION
STEP PutDownWP:
  ACT_PutDownWP(N);
END_STEP
TRANSITION FROM PutDownWP TO SetAutomaticExecuteCompleted
  := WPPutDown;
END_TRANSITION
STEP SetAutomaticExecuteCompleted:
  AutomaticExecuteCompleted(N);
END_STEP
TRANSITION FROM SetAutomaticExecuteCompleted TO Init_ACT_AutomaticExecute
  := AutomaticExecuteCompleted;
END_TRANSITION
END_ACTION

ACTION ACT_EmergencyStop:
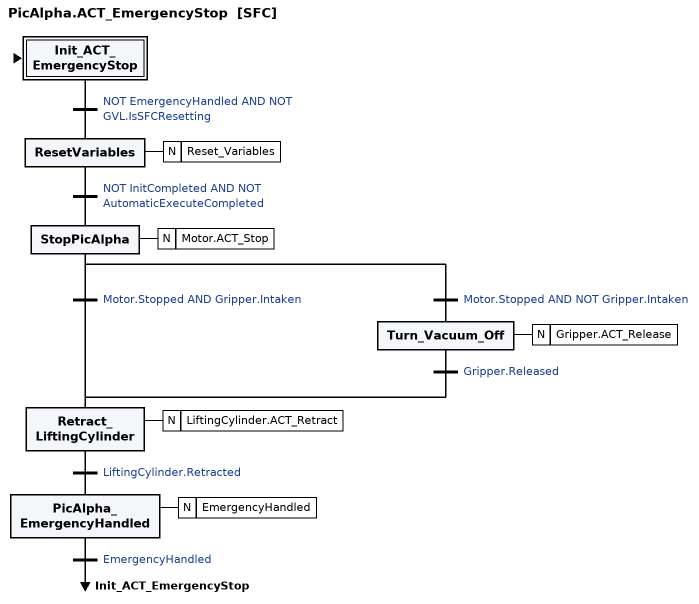
INITIAL_STEP Init_ACT_EmergencyStop:
END_STEP
TRANSITION FROM Init_ACT_EmergencyStop TO ResetVariables
  := NOT EmergencyHandled AND NOT GVL.IsSFCResetting;
END_TRANSITION
STEP ResetVariables:
  Reset_Variables(N);
END_STEP
TRANSITION FROM ResetVariables TO StopPicAlpha
  := NOT InitCompleted AND NOT AutomaticExecuteCompleted;
END_TRANSITION
STEP StopPicAlpha:
  Motor.ACT_Stop(N);
END_STEP
TRANSITION FROM StopPicAlpha TO Retract_LiftingCylinder
  := Motor.Stopped AND Gripper.Intaken;
END_TRANSITION
TRANSITION FROM StopPicAlpha TO Turn_Vacuum_Off
  := Motor.Stopped AND NOT Gripper.Intaken;
END_TRANSITION
STEP Turn_Vacuum_Off:
  Gripper.ACT_Release(N);
END_STEP
TRANSITION FROM Turn_Vacuum_Off TO Retract_LiftingCylinder
  := Gripper.Released;
END_TRANSITION
STEP Retract_LiftingCylinder:
  LiftingCylinder.ACT_Retract(N);
END_STEP
TRANSITION FROM Retract_LiftingCylinder TO PicAlpha_EmergencyHandled
  := LiftingCylinder.Retracted;
END_TRANSITION
STEP PicAlpha_EmergencyHandled:
  EmergencyHandled(N);
END_STEP
TRANSITION FROM PicAlpha_EmergencyHandled TO Init_ACT_EmergencyStop
  := EmergencyHandled;
END_TRANSITION
END_ACTION

ACTION ACT_Init:
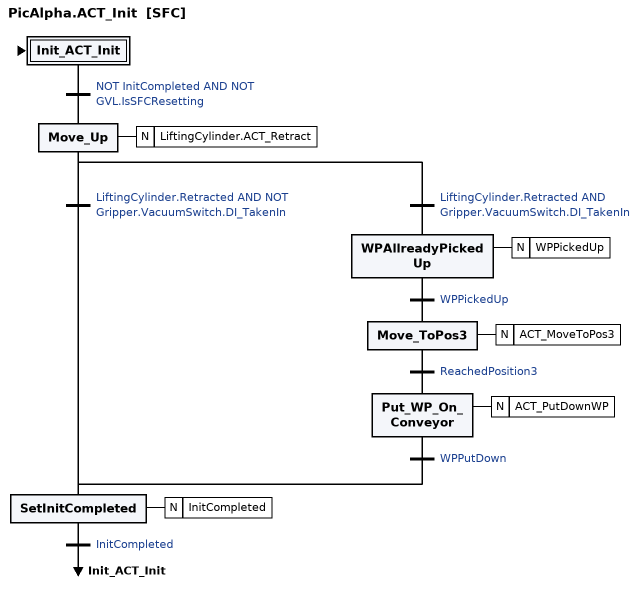
INITIAL_STEP Init_ACT_Init:
END_STEP
TRANSITION FROM Init_ACT_Init TO Move_Up
  := NOT InitCompleted AND NOT GVL.IsSFCResetting;
END_TRANSITION
STEP Move_Up:
  LiftingCylinder.ACT_Retract(N);
END_STEP
TRANSITION FROM Move_Up TO SetInitCompleted
  := LiftingCylinder.Retracted AND NOT Gripper.VacuumSwitch.DI_TakenIn;
END_TRANSITION
TRANSITION FROM Move_Up TO WPAllreadyPickedUp
  := LiftingCylinder.Retracted AND Gripper.VacuumSwitch.DI_TakenIn;
END_TRANSITION
STEP WPAllreadyPickedUp:
  WPPickedUp(N);
END_STEP
TRANSITION FROM WPAllreadyPickedUp TO Move_ToPos3
  := WPPickedUp;
END_TRANSITION
STEP Move_ToPos3:
  ACT_MoveToPos3(N);
END_STEP
TRANSITION FROM Move_ToPos3 TO Put_WP_On_Conveyor
  := ReachedPosition3;
END_TRANSITION
STEP Put_WP_On_Conveyor:
  ACT_PutDownWP(N);
END_STEP
TRANSITION FROM Put_WP_On_Conveyor TO SetInitCompleted
  := WPPutDown;
END_TRANSITION
STEP SetInitCompleted:
  InitCompleted(N);
END_STEP
TRANSITION FROM SetInitCompleted TO Init_ACT_Init
  := InitCompleted;
END_TRANSITION
END_ACTION
END_FUNCTION_BLOCK

FUNCTION_BLOCK RefillConveyor
VAR_INPUT
	//Hardware
	PsBegining : PresenceSensor;
	PsSwitch : PresenceSensor;	
	Switch : Switch;
	Motor : Motor;
	
	//Software	
	Check_AllowedToInit : BOOL;
	Check_AllowedToReceive : BOOL;
	Check_AllowedToSend : BOOL;
	Check_FollowConveyor_InitCompleted : BOOL;
	Check_FollowConveyor_AutomaticExecuteCompleted : BOOL;
	Check_EngineStop: BOOL;
	SFCReset : BOOL;	//Only for SFC implementation
END_VAR
VAR_OUTPUT
	//Software
	InitCompleted : BOOL;
	FollowConveyor_AllowedToInit : BOOL;
	FollowConveyor_AllowedToOperate: BOOL;
	AutomaticExecuteReceivingCompleted : BOOL;
	IsSending : BOOL;
	AutomaticExecuteSendingCompleted : BOOL;
	EmergencyHandled : BOOL;	
END_VAR
VAR
	//Hardware		
	ConveyorSpeed AT %Q* : INT;
	
	//Software
	NumberOfWPs : USINT;
	WPSeperated : BOOL;
END_VAR

                  Check_AllowedToInit := Main.Check_RefillConveyor_AllowedToInit;
Check_AllowedToReceive := Main.Check_RefillConveyor_AllowedToReceive;
Check_AllowedToSend := Main.Check_RefillConveyor_AllowedToSend;
Check_FollowConveyor_InitCompleted := Main.Check_RefillConveyor_FollowConveyor_InitCompleted;
Check_FollowConveyor_AutomaticExecuteCompleted := Main.Check_RefillConveyor_FollowConveyor_AutomaticExecuteCompleted;
Check_EngineStop := MAIN.PPU_EngineStop;
IF Check_EngineStop THEN
	Motor.ACT_Stop();
END_IF
                

ACTION CountUp_WPNumber:
                      NumberOfWPs := NumberOfWPs+1;
                    
END_ACTION

ACTION Reduce_WPNumber:
                      NumberOfWPs := NumberOfWPs-1;
                    
END_ACTION

ACTION Reset_FollowConveyorAllowedToInit:
                      FollowConveyor_AllowedToInit := FALSE;
                    
END_ACTION

ACTION Reset_FollowConveyorAllowedToOperate:
                      FollowConveyor_AllowedToOperate := FALSE;
                    
END_ACTION

ACTION Reset_Variables:
                      InitCompleted := FALSE;
FollowConveyor_AllowedToInit := FALSE;
FollowConveyor_AllowedToOperate := FALSE;
AutomaticExecuteReceivingCompleted := FALSE;
AutomaticExecuteSendingCompleted := FALSE;
NumberOfWPs := 0;
WPSeperated := FALSE;
Check_FollowConveyor_InitCompleted := FALSE;
Check_AllowedToReceive := FALSE;
Check_AllowedToSend := FALSE;
Check_FollowConveyor_AutomaticExecuteCompleted := FALSE;
                    
END_ACTION

ACTION Set_FollowConveyorAllowedToInit:
                      FollowConveyor_AllowedToInit := TRUE;
                    
END_ACTION

ACTION Set_FollowConveyorAllowedToOperate:
                      FollowConveyor_AllowedToOperate := TRUE;
                    
END_ACTION

ACTION ACT_SeperateWP:
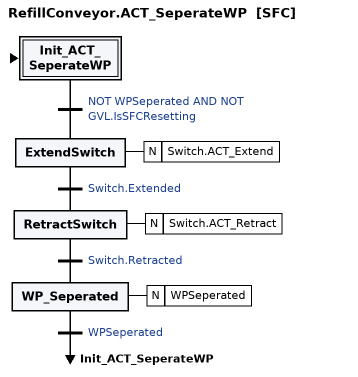
INITIAL_STEP Init_ACT_SeperateWP:
END_STEP
TRANSITION FROM Init_ACT_SeperateWP TO ExtendSwitch
  := NOT WPSeperated AND NOT GVL.IsSFCResetting;
END_TRANSITION
STEP ExtendSwitch:
  Switch.ACT_Extend(N);
END_STEP
TRANSITION FROM ExtendSwitch TO RetractSwitch
  := Switch.Extended;
END_TRANSITION
STEP RetractSwitch:
  Switch.ACT_Retract(N);
END_STEP
TRANSITION FROM RetractSwitch TO WP_Seperated
  := Switch.Retracted;
END_TRANSITION
STEP WP_Seperated:
  WPSeperated(N);
END_STEP
TRANSITION FROM WP_Seperated TO Init_ACT_SeperateWP
  := WPSeperated;
END_TRANSITION
END_ACTION

ACTION ACT_AutomaticExecute:
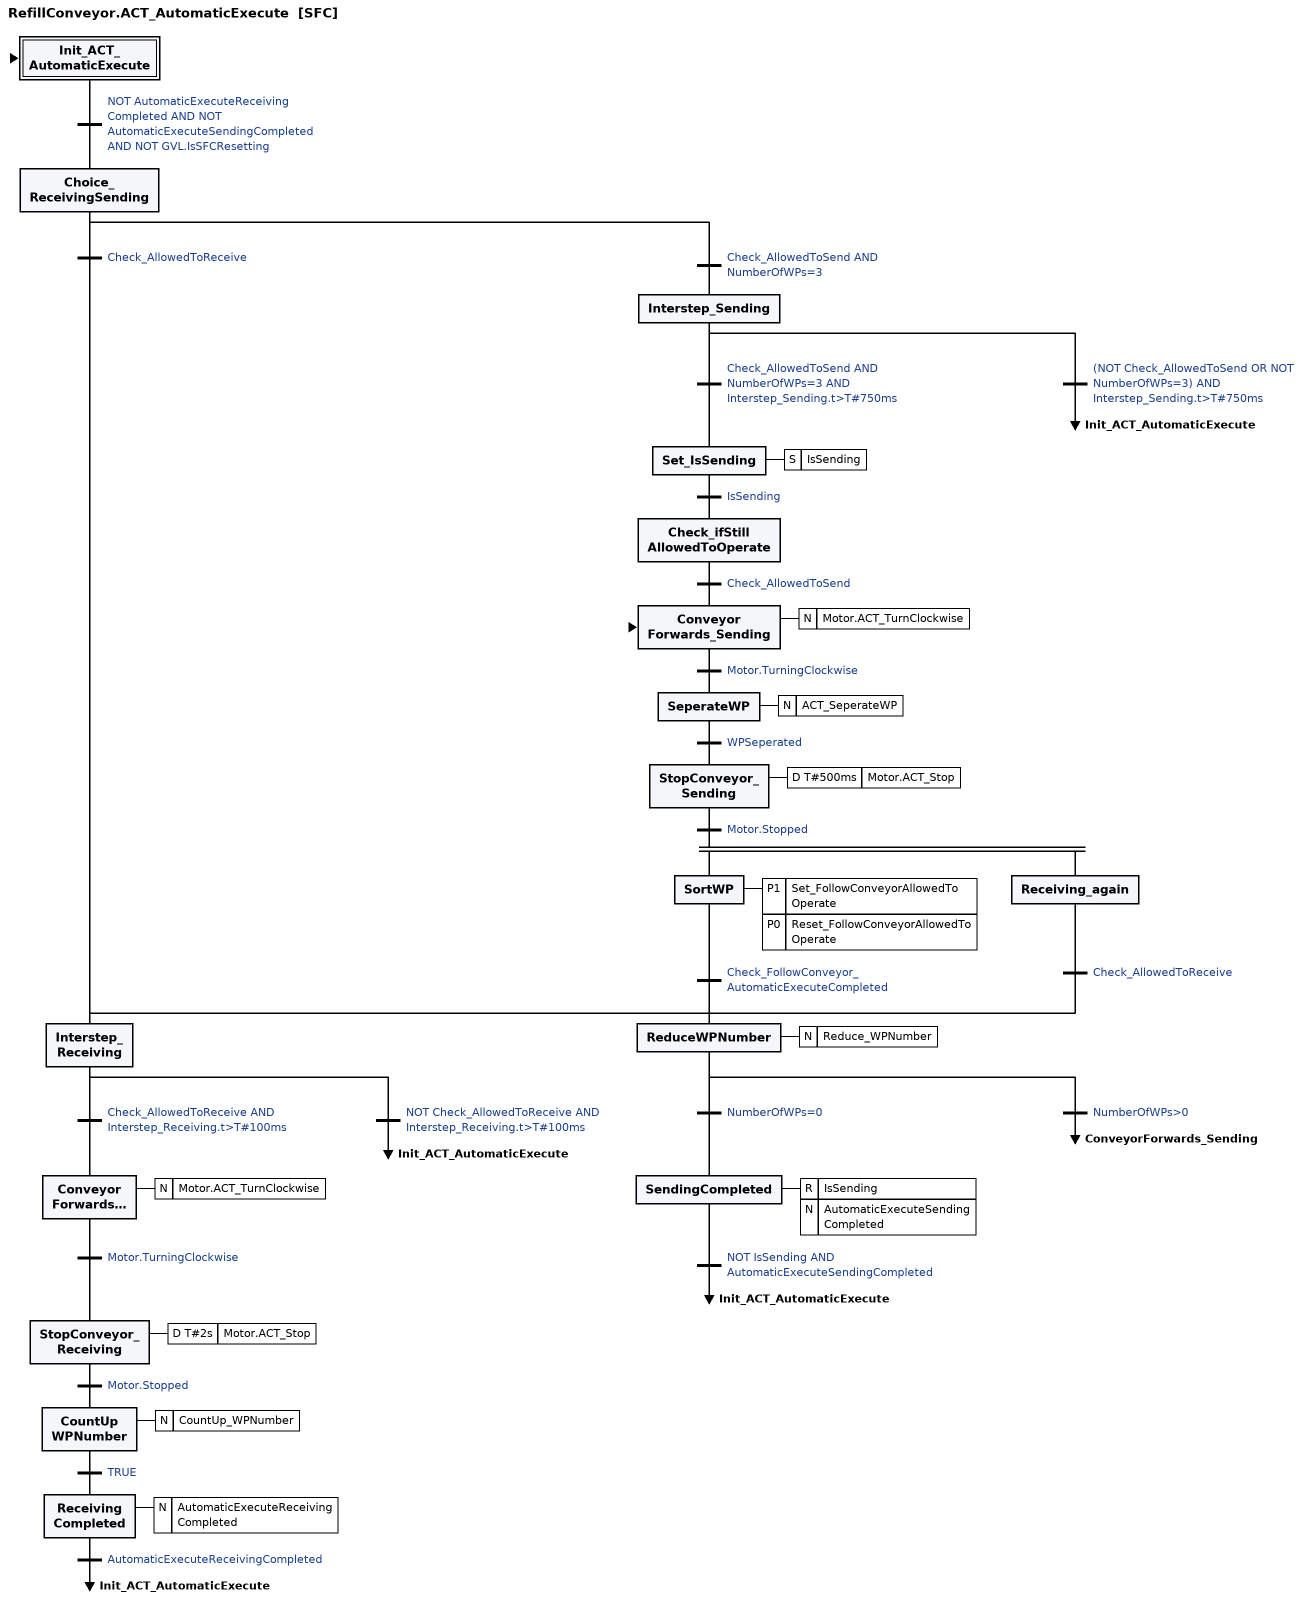
INITIAL_STEP Init_ACT_AutomaticExecute:
END_STEP
TRANSITION FROM Init_ACT_AutomaticExecute TO Choice_ReceivingSending
  := NOT AutomaticExecuteReceivingCompleted AND NOT AutomaticExecuteSendingCompleted AND NOT GVL.IsSFCResetting;
END_TRANSITION
STEP Choice_ReceivingSending:
END_STEP
TRANSITION FROM Choice_ReceivingSending TO Interstep_Receiving
  := Check_AllowedToReceive;
END_TRANSITION
TRANSITION FROM Choice_ReceivingSending TO Interstep_Sending
  := Check_AllowedToSend AND NumberOfWPs=3;
END_TRANSITION
STEP Interstep_Receiving:
END_STEP
TRANSITION FROM Interstep_Receiving TO ConveyorForwards_Receiving
  := Check_AllowedToReceive AND Interstep_Receiving.t>T#100ms;
END_TRANSITION
TRANSITION FROM Interstep_Receiving TO Init_ACT_AutomaticExecute
  := NOT Check_AllowedToReceive AND Interstep_Receiving.t>T#100ms;
END_TRANSITION
STEP ConveyorForwards_Receiving:
  Motor.ACT_TurnClockwise(N);
END_STEP
TRANSITION FROM ConveyorForwards_Receiving TO StopConveyor_Receiving
  := Motor.TurningClockwise;
END_TRANSITION
STEP StopConveyor_Receiving:
  Motor.ACT_Stop(D, T#2s);
END_STEP
TRANSITION FROM StopConveyor_Receiving TO CountUpWPNumber
  := Motor.Stopped;
END_TRANSITION
STEP CountUpWPNumber:
  CountUp_WPNumber(N);
END_STEP
TRANSITION FROM CountUpWPNumber TO ReceivingCompleted
  := TRUE;
END_TRANSITION
STEP ReceivingCompleted:
  AutomaticExecuteReceivingCompleted(N);
END_STEP
TRANSITION FROM ReceivingCompleted TO Init_ACT_AutomaticExecute
  := AutomaticExecuteReceivingCompleted;
END_TRANSITION
STEP Interstep_Sending:
END_STEP
TRANSITION FROM Interstep_Sending TO Set_IsSending
  := Check_AllowedToSend AND NumberOfWPs=3 AND Interstep_Sending.t>T#750ms;
END_TRANSITION
TRANSITION FROM Interstep_Sending TO Init_ACT_AutomaticExecute
  := (NOT Check_AllowedToSend OR NOT NumberOfWPs=3) AND Interstep_Sending.t>T#750ms;
END_TRANSITION
STEP Set_IsSending:
  IsSending(S);
END_STEP
TRANSITION FROM Set_IsSending TO Check_ifStillAllowedToOperate
  := IsSending;
END_TRANSITION
STEP Check_ifStillAllowedToOperate:
END_STEP
TRANSITION FROM Check_ifStillAllowedToOperate TO ConveyorForwards_Sending
  := Check_AllowedToSend;
END_TRANSITION
STEP ConveyorForwards_Sending:
  Motor.ACT_TurnClockwise(N);
END_STEP
TRANSITION FROM ConveyorForwards_Sending TO SeperateWP
  := Motor.TurningClockwise;
END_TRANSITION
STEP SeperateWP:
  ACT_SeperateWP(N);
END_STEP
TRANSITION FROM SeperateWP TO StopConveyor_Sending
  := WPSeperated;
END_TRANSITION
STEP StopConveyor_Sending:
  Motor.ACT_Stop(D, T#500ms);
END_STEP
TRANSITION FROM StopConveyor_Sending TO (SortWP, Receiving_again)
  := Motor.Stopped;
END_TRANSITION
STEP SortWP:
  Set_FollowConveyorAllowedToOperate(P1);
  Reset_FollowConveyorAllowedToOperate(P0);
END_STEP
TRANSITION FROM SortWP TO ReduceWPNumber
  := Check_FollowConveyor_AutomaticExecuteCompleted;
END_TRANSITION
STEP Receiving_again:
END_STEP
TRANSITION FROM Receiving_again TO Interstep_Receiving
  := Check_AllowedToReceive;
END_TRANSITION
STEP ReduceWPNumber:
  Reduce_WPNumber(N);
END_STEP
TRANSITION FROM ReduceWPNumber TO SendingCompleted
  := NumberOfWPs=0;
END_TRANSITION
TRANSITION FROM ReduceWPNumber TO ConveyorForwards_Sending
  := NumberOfWPs>0;
END_TRANSITION
STEP SendingCompleted:
  IsSending(R);
  AutomaticExecuteSendingCompleted(N);
END_STEP
TRANSITION FROM SendingCompleted TO Init_ACT_AutomaticExecute
  := NOT IsSending AND AutomaticExecuteSendingCompleted;
END_TRANSITION
END_ACTION

ACTION ACT_EmergencyStop:
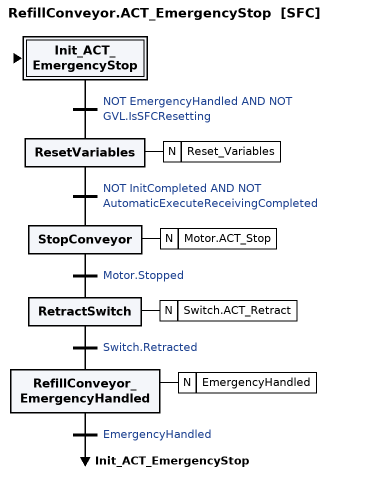
INITIAL_STEP Init_ACT_EmergencyStop:
END_STEP
TRANSITION FROM Init_ACT_EmergencyStop TO ResetVariables
  := NOT EmergencyHandled AND NOT GVL.IsSFCResetting;
END_TRANSITION
STEP ResetVariables:
  Reset_Variables(N);
END_STEP
TRANSITION FROM ResetVariables TO StopConveyor
  := NOT InitCompleted AND NOT AutomaticExecuteReceivingCompleted;
END_TRANSITION
STEP StopConveyor:
  Motor.ACT_Stop(N);
END_STEP
TRANSITION FROM StopConveyor TO RetractSwitch
  := Motor.Stopped;
END_TRANSITION
STEP RetractSwitch:
  Switch.ACT_Retract(N);
END_STEP
TRANSITION FROM RetractSwitch TO RefillConveyor_EmergencyHandled
  := Switch.Retracted;
END_TRANSITION
STEP RefillConveyor_EmergencyHandled:
  EmergencyHandled(N);
END_STEP
TRANSITION FROM RefillConveyor_EmergencyHandled TO Init_ACT_EmergencyStop
  := EmergencyHandled;
END_TRANSITION
END_ACTION

ACTION ACT_Init:
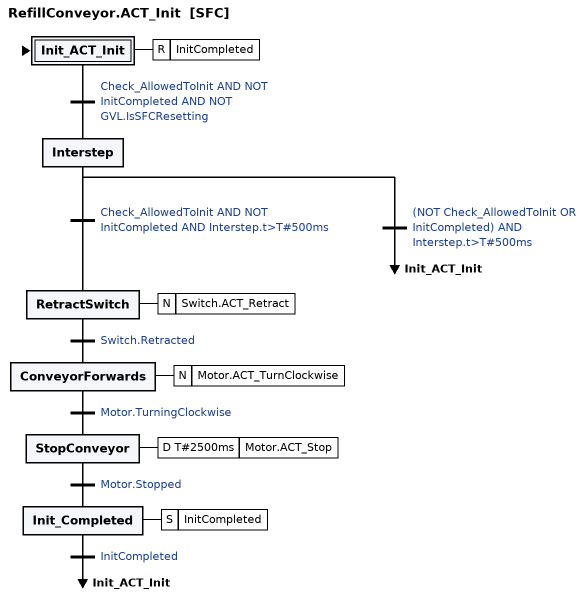
INITIAL_STEP Init_ACT_Init:
  InitCompleted(R);
END_STEP
TRANSITION FROM Init_ACT_Init TO Interstep
  := Check_AllowedToInit AND NOT InitCompleted AND NOT GVL.IsSFCResetting;
END_TRANSITION
STEP Interstep:
END_STEP
TRANSITION FROM Interstep TO RetractSwitch
  := Check_AllowedToInit AND NOT InitCompleted AND Interstep.t>T#500ms;
END_TRANSITION
TRANSITION FROM Interstep TO Init_ACT_Init
  := (NOT Check_AllowedToInit OR InitCompleted) AND Interstep.t>T#500ms;
END_TRANSITION
STEP RetractSwitch:
  Switch.ACT_Retract(N);
END_STEP
TRANSITION FROM RetractSwitch TO ConveyorForwards
  := Switch.Retracted;
END_TRANSITION
STEP ConveyorForwards:
  Motor.ACT_TurnClockwise(N);
END_STEP
TRANSITION FROM ConveyorForwards TO StopConveyor
  := Motor.TurningClockwise;
END_TRANSITION
STEP StopConveyor:
  Motor.ACT_Stop(D, T#2500ms);
END_STEP
TRANSITION FROM StopConveyor TO Init_Completed
  := Motor.Stopped;
END_TRANSITION
STEP Init_Completed:
  InitCompleted(S);
END_STEP
TRANSITION FROM Init_Completed TO Init_ACT_Init
  := InitCompleted;
END_TRANSITION
END_ACTION
END_FUNCTION_BLOCK

FUNCTION_BLOCK PicAlphaConveyor
VAR_INPUT
	//Hardware
	PsSwitch : PresenceSensor;
	PsEnd : PresenceSensor;
	Switch : Switch;
	Motor : Motor;
	
	//Software	
	Check_AllowedToInit : BOOL;
	Check_AllowedToReceive : BOOL;
	Check_AllowedToSend : BOOL;
	Check_FollowConveyor_InitCompleted : BOOL;
	Check_PicAlpha_AutomaticExecuteCompleted : BOOL;
	Check_FollowConveyor_AutomaticExecuteCompleted : BOOL;	
	Check_EngineStop: BOOL;
	SFCReset : BOOL;	//Only for SFC implementation
END_VAR
VAR_OUTPUT
	//Software
	InitCompleted : BOOL;
	FollowConveyor_AllowedToInit : BOOL;
	PicAlpha_AllowedToOperate : BOOL;
	FollowConveyor_AllowedToOperate: BOOL;
	AutomaticExecuteReceivingCompleted : BOOL;
	AutomaticExecuteSendingCompleted : BOOL;
	EmergencyHandled : BOOL;	
END_VAR
VAR
	//Hardware		
	ConveyorSpeed AT %Q* : INT;
	
	//Software
	NumberOfWPs : INT;
	WPSeperated : BOOL;
END_VAR

                  Check_AllowedToInit := Main.Check_PicAlphaConveyor_AllowedToInit;
Check_AllowedToReceive := Main.Check_PicAlphaConveyor_AllowedToReceive;
Check_AllowedToSend := Main.Check_PicAlphaConveyor_AllowedToSend;
Check_FollowConveyor_InitCompleted := Main.Check_PicAlphaConveyor_FollowConveyor_InitCompleted;
Check_PicAlpha_AutomaticExecuteCompleted := Main.Check_PicAlphaConveyor_PicAlpha_AutomaticExecuteCompleted;
Check_FollowConveyor_AutomaticExecuteCompleted := Main.Check_PicAlphaConveyor_FollowConveyor_AutomaticExecuteCompleted;
Check_EngineStop := MAIN.PPU_EngineStop;
IF Check_EngineStop THEN
	Motor.ACT_Stop();
END_IF
                

ACTION Reduce_WPNumber:
                      NumberOfWPs := NumberOfWPs-1;
                    
END_ACTION

ACTION Reset_FollowConveyorAllowedToInit:
                      FollowConveyor_AllowedToInit := FALSE;
                    
END_ACTION

ACTION Reset_FollowConveyorAllowedToOperate:
                      FollowConveyor_AllowedToOperate := FALSE;
                    
END_ACTION

ACTION Reset_Variables:
                      InitCompleted := FALSE;
FollowConveyor_AllowedToInit := FALSE;
PicAlpha_AllowedToOperate := FALSE;
FollowConveyor_AllowedToOperate := FALSE;
AutomaticExecuteReceivingCompleted := FALSE;
AutomaticExecuteSendingCompleted := FALSE;

NumberOfWPs := 0;
WPSeperated := FALSE;
                    
END_ACTION

ACTION Rest_PicAlpha_AllowedToOperate:
                      PicAlpha_AllowedToOperate := FALSE;
                    
END_ACTION

ACTION Set_FollowConveyorAllowedToInit:
                      FollowConveyor_AllowedToInit := TRUE;
                    
END_ACTION

ACTION Set_FollowConveyorAllowedToOperate:
                      FollowConveyor_AllowedToOperate := TRUE;
                    
END_ACTION

ACTION Set_NumberOfWPsTo3:
                      NumberOfWPs := 3;
                    
END_ACTION

ACTION Set_PicAlpha_AllowedToOperate:
                      PicAlpha_AllowedToOperate := TRUE;
                    
END_ACTION

ACTION ACT_SeperateWP:
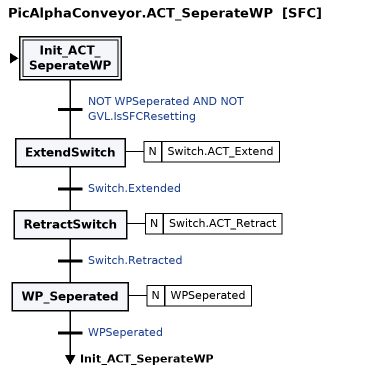
INITIAL_STEP Init_ACT_SeperateWP:
END_STEP
TRANSITION FROM Init_ACT_SeperateWP TO ExtendSwitch
  := NOT WPSeperated AND NOT GVL.IsSFCResetting;
END_TRANSITION
STEP ExtendSwitch:
  Switch.ACT_Extend(N);
END_STEP
TRANSITION FROM ExtendSwitch TO RetractSwitch
  := Switch.Extended;
END_TRANSITION
STEP RetractSwitch:
  Switch.ACT_Retract(N);
END_STEP
TRANSITION FROM RetractSwitch TO WP_Seperated
  := Switch.Retracted;
END_TRANSITION
STEP WP_Seperated:
  WPSeperated(N);
END_STEP
TRANSITION FROM WP_Seperated TO Init_ACT_SeperateWP
  := WPSeperated;
END_TRANSITION
END_ACTION

ACTION ACT_AutomaticExecute:
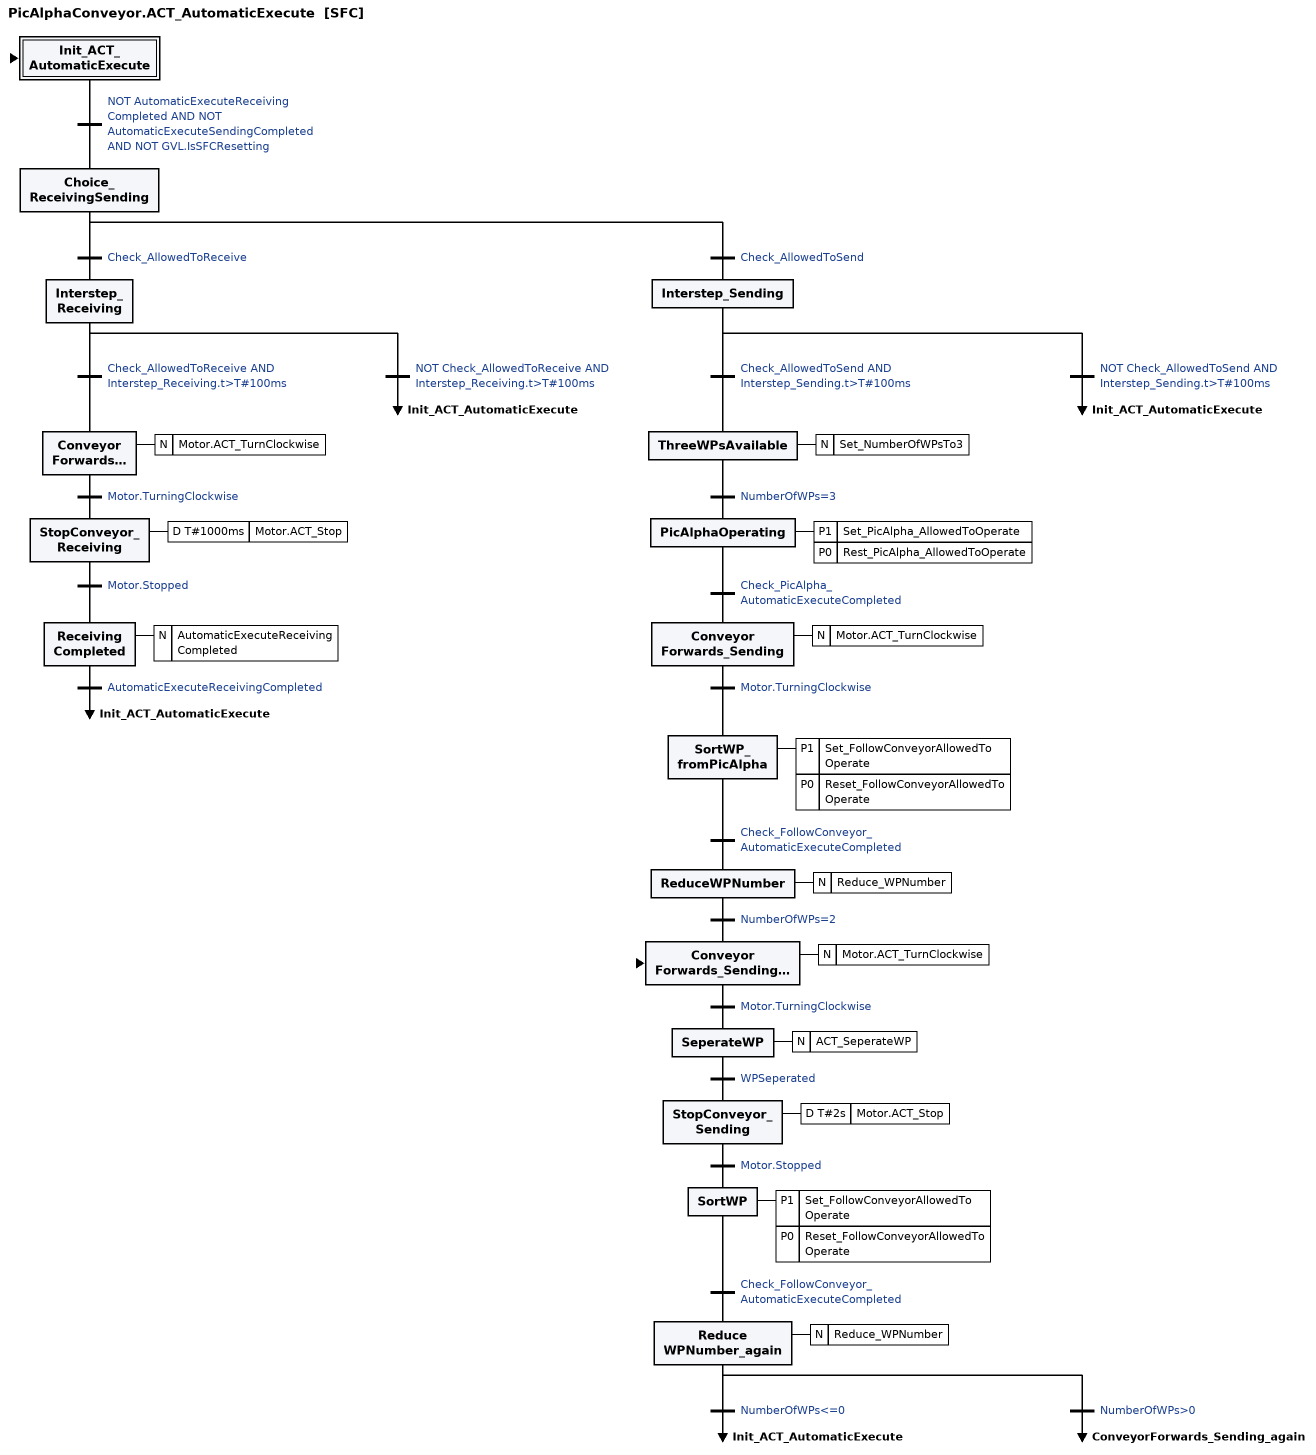
INITIAL_STEP Init_ACT_AutomaticExecute:
END_STEP
TRANSITION FROM Init_ACT_AutomaticExecute TO Choice_ReceivingSending
  := NOT AutomaticExecuteReceivingCompleted AND NOT AutomaticExecuteSendingCompleted AND NOT GVL.IsSFCResetting;
END_TRANSITION
STEP Choice_ReceivingSending:
END_STEP
TRANSITION FROM Choice_ReceivingSending TO Interstep_Receiving
  := Check_AllowedToReceive;
END_TRANSITION
TRANSITION FROM Choice_ReceivingSending TO Interstep_Sending
  := Check_AllowedToSend;
END_TRANSITION
STEP Interstep_Receiving:
END_STEP
TRANSITION FROM Interstep_Receiving TO ConveyorForwards_Receiving
  := Check_AllowedToReceive AND Interstep_Receiving.t>T#100ms;
END_TRANSITION
TRANSITION FROM Interstep_Receiving TO Init_ACT_AutomaticExecute
  := NOT Check_AllowedToReceive AND Interstep_Receiving.t>T#100ms;
END_TRANSITION
STEP ConveyorForwards_Receiving:
  Motor.ACT_TurnClockwise(N);
END_STEP
TRANSITION FROM ConveyorForwards_Receiving TO StopConveyor_Receiving
  := Motor.TurningClockwise;
END_TRANSITION
STEP StopConveyor_Receiving:
  Motor.ACT_Stop(D, T#1000ms);
END_STEP
TRANSITION FROM StopConveyor_Receiving TO ReceivingCompleted
  := Motor.Stopped;
END_TRANSITION
STEP ReceivingCompleted:
  AutomaticExecuteReceivingCompleted(N);
END_STEP
TRANSITION FROM ReceivingCompleted TO Init_ACT_AutomaticExecute
  := AutomaticExecuteReceivingCompleted;
END_TRANSITION
STEP Interstep_Sending:
END_STEP
TRANSITION FROM Interstep_Sending TO ThreeWPsAvailable
  := Check_AllowedToSend AND Interstep_Sending.t>T#100ms;
END_TRANSITION
TRANSITION FROM Interstep_Sending TO Init_ACT_AutomaticExecute
  := NOT Check_AllowedToSend AND Interstep_Sending.t>T#100ms;
END_TRANSITION
STEP ThreeWPsAvailable:
  Set_NumberOfWPsTo3(N);
END_STEP
TRANSITION FROM ThreeWPsAvailable TO PicAlphaOperating
  := NumberOfWPs=3;
END_TRANSITION
STEP PicAlphaOperating:
  Set_PicAlpha_AllowedToOperate(P1);
  Rest_PicAlpha_AllowedToOperate(P0);
END_STEP
TRANSITION FROM PicAlphaOperating TO ConveyorForwards_Sending
  := Check_PicAlpha_AutomaticExecuteCompleted;
END_TRANSITION
STEP ConveyorForwards_Sending:
  Motor.ACT_TurnClockwise(N);
END_STEP
TRANSITION FROM ConveyorForwards_Sending TO SortWP_fromPicAlpha
  := Motor.TurningClockwise;
END_TRANSITION
STEP SortWP_fromPicAlpha:
  Set_FollowConveyorAllowedToOperate(P1);
  Reset_FollowConveyorAllowedToOperate(P0);
END_STEP
TRANSITION FROM SortWP_fromPicAlpha TO ReduceWPNumber
  := Check_FollowConveyor_AutomaticExecuteCompleted;
END_TRANSITION
STEP ReduceWPNumber:
  Reduce_WPNumber(N);
END_STEP
TRANSITION FROM ReduceWPNumber TO ConveyorForwards_Sending_again
  := NumberOfWPs=2;
END_TRANSITION
STEP ConveyorForwards_Sending_again:
  Motor.ACT_TurnClockwise(N);
END_STEP
TRANSITION FROM ConveyorForwards_Sending_again TO SeperateWP
  := Motor.TurningClockwise;
END_TRANSITION
STEP SeperateWP:
  ACT_SeperateWP(N);
END_STEP
TRANSITION FROM SeperateWP TO StopConveyor_Sending
  := WPSeperated;
END_TRANSITION
STEP StopConveyor_Sending:
  Motor.ACT_Stop(D, T#2s);
END_STEP
TRANSITION FROM StopConveyor_Sending TO SortWP
  := Motor.Stopped;
END_TRANSITION
STEP SortWP:
  Set_FollowConveyorAllowedToOperate(P1);
  Reset_FollowConveyorAllowedToOperate(P0);
END_STEP
TRANSITION FROM SortWP TO ReduceWPNumber_again
  := Check_FollowConveyor_AutomaticExecuteCompleted;
END_TRANSITION
STEP ReduceWPNumber_again:
  Reduce_WPNumber(N);
END_STEP
TRANSITION FROM ReduceWPNumber_again TO Init_ACT_AutomaticExecute
  := NumberOfWPs<=0;
END_TRANSITION
TRANSITION FROM ReduceWPNumber_again TO ConveyorForwards_Sending_again
  := NumberOfWPs>0;
END_TRANSITION
END_ACTION

ACTION ACT_EmergencyStop:
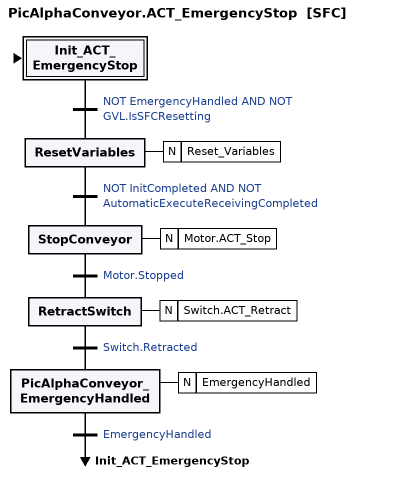
INITIAL_STEP Init_ACT_EmergencyStop:
END_STEP
TRANSITION FROM Init_ACT_EmergencyStop TO ResetVariables
  := NOT EmergencyHandled AND NOT GVL.IsSFCResetting;
END_TRANSITION
STEP ResetVariables:
  Reset_Variables(N);
END_STEP
TRANSITION FROM ResetVariables TO StopConveyor
  := NOT InitCompleted AND NOT AutomaticExecuteReceivingCompleted;
END_TRANSITION
STEP StopConveyor:
  Motor.ACT_Stop(N);
END_STEP
TRANSITION FROM StopConveyor TO RetractSwitch
  := Motor.Stopped;
END_TRANSITION
STEP RetractSwitch:
  Switch.ACT_Retract(N);
END_STEP
TRANSITION FROM RetractSwitch TO PicAlphaConveyor_EmergencyHandled
  := Switch.Retracted;
END_TRANSITION
STEP PicAlphaConveyor_EmergencyHandled:
  EmergencyHandled(N);
END_STEP
TRANSITION FROM PicAlphaConveyor_EmergencyHandled TO Init_ACT_EmergencyStop
  := EmergencyHandled;
END_TRANSITION
END_ACTION

ACTION ACT_Init:
